  MoveL 3264 to (40.1, 47.39, -201.09) mm, rotated rx -152.51 ry -6.42 rz -112.51 deg; joints [11.465, -29.015, 82.683, 214.408, 104.039, 41.667, 26.033]
  MoveL 3265 to (39.93, 47.72, -201.04) mm, rotated rx -152.51 ry -6.42 rz -112.51 deg; joints [11.469, -29.014, 82.657, 214.407, 104.02, 41.65, 26.033]
  MoveL 3266 to (39.8, 48.12, -201) mm, rotated rx -152.51 ry -6.42 rz -112.51 deg; joints [11.471, -29.013, 82.629, 214.404, 103.997, 41.633, 26.033]
  MoveL 3267 to (39.72, 48.56, -200.98) mm, rotated rx -152.51 ry -6.42 rz -112.51 deg; joints [11.471, -29.014, 82.599, 214.4, 103.972, 41.615, 26.033]
  MoveL 3268 to (39.68, 49.06, -200.97) mm, rotated rx -152.51 ry -6.42 rz -112.51 deg; joints [11.47, -29.015, 82.566, 214.394, 103.943, 41.596, 26.033]
  MoveL 3269 to (39.66, 49.57, -200.97) mm, rotated rx -152.51 ry -6.42 rz -112.51 deg; joints [11.467, -29.017, 82.533, 214.388, 103.914, 41.577, 26.033]
  MoveL 3270 to (39.65, 50.63, -200.97) mm, rotated rx -152.51 ry -6.42 rz -112.51 deg; joints [11.461, -29.02, 82.466, 214.374, 103.854, 41.539, 26.033]
  MoveL 3271 to (39.63, 51.12, -200.95) mm, rotated rx -152.51 ry -6.42 rz -112.51 deg; joints [11.459, -29.021, 82.433, 214.368, 103.826, 41.52, 26.033]
  MoveL 3272 to (39.59, 51.58, -200.9) mm, rotated rx -152.51 ry -6.42 rz -112.51 deg; joints [11.458, -29.019, 82.399, 214.362, 103.798, 41.502, 26.033]
  MoveL 3273 to (39.53, 52.1, -200.82) mm, rotated rx -152.51 ry -6.42 rz -112.51 deg; joints [11.457, -29.016, 82.358, 214.357, 103.767, 41.481, 26.033]
  MoveL 3274 to (39.48, 52.68, -200.76) mm, rotated rx -152.51 ry -6.42 rz -112.51 deg; joints [11.456, -29.013, 82.315, 214.35, 103.733, 41.458, 26.033]
  MoveL 3275 to (39.45, 53.26, -200.73) mm, rotated rx -152.51 ry -6.42 rz -112.51 deg; joints [11.453, -29.013, 82.275, 214.343, 103.7, 41.436, 26.033]
  MoveL 3276 to (39.44, 53.79, -200.71) mm, rotated rx -152.51 ry -6.42 rz -112.51 deg; joints [11.45, -29.013, 82.239, 214.336, 103.669, 41.416, 26.033]
  MoveL 3277 to (39.43, 54.33, -200.71) mm, rotated rx -152.51 ry -6.42 rz -112.51 deg; joints [11.448, -29.015, 82.204, 214.329, 103.638, 41.397, 26.033]
  MoveL 3278 to (39.42, 55.38, -200.71) mm, rotated rx -152.51 ry -6.42 rz -112.51 deg; joints [11.442, -29.018, 82.137, 214.316, 103.578, 41.359, 26.033]
  MoveL 3279 to (39.37, 56.41, -200.69) mm, rotated rx -152.51 ry -6.42 rz -112.51 deg; joints [11.437, -29.019, 82.069, 214.303, 103.519, 41.321, 26.033]
  MoveL 3280 to (39.34, 59.03, -200.69) mm, rotated rx -152.51 ry -6.42 rz -112.51 deg; joints [11.423, -29.026, 81.9, 214.27, 103.369, 41.227, 26.033]
  MoveL 3281 to (39.39, 60.47, -200.77) mm, rotated rx -152.51 ry -6.42 rz -112.51 deg; joints [11.412, -29.035, 81.815, 214.25, 103.288, 41.178, 26.033]
  MoveL 3282 to (39.58, 61.64, -201.04) mm, rotated rx -152.51 ry -6.42 rz -112.51 deg; joints [11.398, -29.054, 81.764, 214.231, 103.225, 41.145, 26.033]
  MoveL 3283 to (39.9, 62.52, -201.47) mm, rotated rx -152.51 ry -6.42 rz -112.51 deg; joints [11.38, -29.083, 81.749, 214.213, 103.182, 41.128, 26.033]
  MoveL 3284 to (40.12, 62.85, -201.76) mm, rotated rx -152.51 ry -6.42 rz -112.51 deg; joints [11.37, -29.102, 81.754, 214.204, 103.168, 41.126, 26.033]
  MoveL 3285 to (40.37, 63.12, -202.09) mm, rotated rx -152.51 ry -6.42 rz -112.51 deg; joints [11.359, -29.123, 81.768, 214.196, 103.158, 41.128, 26.033]
  MoveL 3286 to (40.97, 63.44, -202.88) mm, rotated rx -152.51 ry -6.42 rz -112.51 deg; joints [11.334, -29.173, 81.823, 214.179, 103.153, 41.143, 26.033]
  MoveL 3287 to (41.71, 63.48, -203.84) mm, rotated rx -152.51 ry -6.42 rz -112.51 deg; joints [11.305, -29.234, 81.912, 214.164, 103.167, 41.174, 26.033]
  MoveL 3288 to (43.6, 62.7, -206.3) mm, rotated rx -152.51 ry -6.42 rz -112.51 deg; joints [11.236, -29.386, 82.195, 214.134, 103.252, 41.285, 26.033]
  MoveL 3289 to (45.46, 61.14, -208.75) mm, rotated rx -152.51 ry -6.42 rz -112.51 deg; joints [11.173, -29.535, 82.528, 214.116, 103.383, 41.423, 26.033]
  MoveL 3290 to (46.69, 59.12, -210.51) mm, rotated rx -152.51 ry -6.42 rz -112.51 deg; joints [11.137, -29.64, 82.823, 214.117, 103.527, 41.551, 26.033]
  MoveL 3291 to (47.06, 57.94, -211.12) mm, rotated rx -152.51 ry -6.42 rz -112.51 deg; joints [11.129, -29.676, 82.957, 214.124, 103.605, 41.612, 26.033]
  MoveL 3292 to (47.28, 56.65, -211.56) mm, rotated rx -152.51 ry -6.42 rz -112.51 deg; joints [11.127, -29.701, 83.081, 214.137, 103.687, 41.67, 26.033]
  MoveL 3293 to (47.24, 53.72, -211.91) mm, rotated rx -152.51 ry -6.42 rz -112.51 deg; joints [11.144, -29.717, 83.301, 214.176, 103.862, 41.78, 26.033]
  MoveL 3294 to (46.95, 51.11, -211.91) mm, rotated rx -152.51 ry -6.42 rz -112.51 deg; joints [11.169, -29.712, 83.467, 214.217, 104.012, 41.867, 26.033]
  MoveL 3295 to (46.88, 50.59, -211.9) mm, rotated rx -152.51 ry -6.42 rz -112.51 deg; joints [11.174, -29.71, 83.5, 214.226, 104.042, 41.884, 26.033]
  MoveL 3296 to (46.8, 50.05, -211.87) mm, rotated rx -152.51 ry -6.42 rz -112.51 deg; joints [11.18, -29.707, 83.531, 214.235, 104.073, 41.901, 26.033]
  MoveL 3297 to (46.74, 49.56, -211.86) mm, rotated rx -152.51 ry -6.42 rz -112.51 deg; joints [11.185, -29.705, 83.561, 214.243, 104.101, 41.917, 26.033]
  MoveL 3298 to (46.7, 49.11, -211.88) mm, rotated rx -152.51 ry -6.42 rz -112.51 deg; joints [11.189, -29.705, 83.591, 214.249, 104.127, 41.932, 26.033]
  MoveL 3299 to (46.66, 48.63, -211.9) mm, rotated rx -152.51 ry -6.42 rz -112.51 deg; joints [11.193, -29.706, 83.625, 214.257, 104.155, 41.949, 26.033]
  MoveL 3300 to (46.64, 48.05, -211.97) mm, rotated rx -152.51 ry -6.42 rz -112.51 deg; joints [11.197, -29.709, 83.668, 214.265, 104.19, 41.97, 26.033]
  MoveL 3301 to (46.63, 47.47, -212.05) mm, rotated rx -152.51 ry -6.42 rz -112.51 deg; joints [11.2, -29.712, 83.711, 214.273, 104.224, 41.992, 26.033]
  MoveL 3302 to (46.6, 46.9, -212.1) mm, rotated rx -152.51 ry -6.42 rz -112.51 deg; joints [11.204, -29.714, 83.752, 214.282, 104.257, 42.013, 26.033]
  MoveL 3303 to (46.56, 46.37, -212.12) mm, rotated rx -152.51 ry -6.42 rz -112.51 deg; joints [11.209, -29.714, 83.787, 214.29, 104.288, 42.031, 26.033]
  MoveL 3304 to (46.5, 45.86, -212.13) mm, rotated rx -152.51 ry -6.42 rz -112.51 deg; joints [11.214, -29.713, 83.821, 214.298, 104.318, 42.048, 26.033]
  MoveL 3305 to (46.45, 45.34, -212.13) mm, rotated rx -152.51 ry -6.42 rz -112.51 deg; joints [11.219, -29.712, 83.854, 214.306, 104.348, 42.066, 26.033]
  MoveL 3306 to (46.41, 44.77, -212.16) mm, rotated rx -152.51 ry -6.42 rz -112.51 deg; joints [11.223, -29.712, 83.892, 214.315, 104.381, 42.086, 26.033]
  MoveL 3307 to (46.39, 44.22, -212.22) mm, rotated rx -152.51 ry -6.42 rz -112.51 deg; joints [11.227, -29.714, 83.932, 214.323, 104.413, 42.106, 26.033]
  MoveL 3308 to (46.39, 43.66, -212.29) mm, rotated rx -152.51 ry -6.42 rz -112.51 deg; joints [11.23, -29.717, 83.973, 214.331, 104.446, 42.127, 26.033]
  MoveL 3309 to (46.45, 43.16, -212.35) mm, rotated rx -152.51 ry -6.42 rz -112.51 deg; joints [11.231, -29.718, 84.01, 214.336, 104.476, 42.147, 26.033]
  MoveL 3310 to (46.54, 42.71, -212.38) mm, rotated rx -152.51 ry -6.42 rz -112.51 deg; joints [11.23, -29.718, 84.041, 214.341, 104.502, 42.166, 26.033]
  MoveL 3311 to (46.68, 42.33, -212.39) mm, rotated rx -152.51 ry -6.42 rz -112.51 deg; joints [11.227, -29.715, 84.066, 214.343, 104.523, 42.183, 26.033]
  MoveL 3312 to (46.84, 41.98, -212.39) mm, rotated rx -152.51 ry -6.42 rz -112.51 deg; joints [11.224, -29.712, 84.087, 214.344, 104.542, 42.199, 26.033]
  MoveL 3313 to (46.45, 43.21, -213.26) mm, rotated rx -152.51 ry -6.42 rz -112.51 deg; joints [11.226, -29.782, 84.094, 214.336, 104.491, 42.161, 26.033]
  MoveL 3314 to (47.29, 41.84, -213.54) mm, rotated rx -152.51 ry -6.42 rz -112.51 deg; joints [11.205, -29.787, 84.204, 214.337, 104.57, 42.233, 26.033]
  MoveL 3315 to (48.19, 40.28, -213.74) mm, rotated rx -152.51 ry -6.42 rz -112.51 deg; joints [11.183, -29.785, 84.318, 214.339, 104.66, 42.311, 26.033]
  MoveL 3316 to (49.17, 38.48, -213.87) mm, rotated rx -152.51 ry -6.42 rz -112.51 deg; joints [11.161, -29.777, 84.441, 214.343, 104.761, 42.399, 26.033]
  MoveL 3317 to (50.22, 36.49, -213.96) mm, rotated rx -152.51 ry -6.42 rz -112.51 deg; joints [11.137, -29.763, 84.571, 214.348, 104.871, 42.494, 26.033]
  MoveL 3318 to (51.24, 34.61, -214.11) mm, rotated rx -152.51 ry -6.42 rz -112.51 deg; joints [11.114, -29.754, 84.699, 214.353, 104.976, 42.586, 26.033]
  MoveL 3319 to (52.26, 32.73, -214.32) mm, rotated rx -152.51 ry -6.42 rz -112.51 deg; joints [11.09, -29.749, 84.832, 214.357, 105.083, 42.678, 26.033]
  MoveL 3320 to (53.22, 30.94, -214.44) mm, rotated rx -152.51 ry -6.42 rz -112.51 deg; joints [11.068, -29.739, 84.951, 214.362, 105.183, 42.765, 26.033]
  MoveL 3321 to (54.11, 29.32, -214.71) mm, rotated rx -152.51 ry -6.42 rz -112.51 deg; joints [11.046, -29.739, 85.073, 214.365, 105.276, 42.846, 26.033]
  MoveL 3322 to (55.08, 27.5, -214.92) mm, rotated rx -152.51 ry -6.42 rz -112.51 deg; joints [11.024, -29.735, 85.202, 214.37, 105.379, 42.935, 26.033]
  MoveL 3323 to (56.05, 25.66, -215.06) mm, rotated rx -152.51 ry -6.42 rz -112.51 deg; joints [11.001, -29.724, 85.325, 214.375, 105.482, 43.024, 26.033]
  MoveL 3324 to (57.04, 23.77, -215.17) mm, rotated rx -152.51 ry -6.42 rz -112.51 deg; joints [10.979, -29.71, 85.447, 214.381, 105.587, 43.115, 26.033]
  MoveL 3325 to (58.04, 21.89, -215.4) mm, rotated rx -152.51 ry -6.42 rz -112.51 deg; joints [10.956, -29.705, 85.579, 214.387, 105.693, 43.207, 26.033]
  MoveL 3326 to (59.01, 19.98, -215.66) mm, rotated rx -152.51 ry -6.42 rz -112.51 deg; joints [10.933, -29.701, 85.716, 214.393, 105.802, 43.3, 26.033]
  MoveL 3327 to (59.99, 18.09, -215.74) mm, rotated rx -152.51 ry -6.42 rz -112.51 deg; joints [10.911, -29.685, 85.835, 214.399, 105.906, 43.39, 26.033]
  MoveL 3328 to (60.99, 16.16, -215.79) mm, rotated rx -152.51 ry -6.42 rz -112.51 deg; joints [10.888, -29.666, 85.952, 214.406, 106.012, 43.481, 26.033]
  MoveL 3329 to (61.95, 14.28, -215.89) mm, rotated rx -152.51 ry -6.42 rz -112.51 deg; joints [10.867, -29.651, 86.071, 214.412, 106.116, 43.57, 26.033]
  MoveL 3330 to (62.91, 12.39, -216.1) mm, rotated rx -152.51 ry -6.42 rz -112.51 deg; joints [10.844, -29.642, 86.2, 214.419, 106.222, 43.662, 26.033]
  MoveL 3331 to (63.84, 10.53, -216.43) mm, rotated rx -152.51 ry -6.42 rz -112.51 deg; joints [10.822, -29.642, 86.338, 214.426, 106.329, 43.753, 26.033]
  MoveL 3332 to (64.79, 8.6, -216.69) mm, rotated rx -152.51 ry -6.42 rz -112.51 deg; joints [10.801, -29.637, 86.474, 214.435, 106.439, 43.847, 26.033]
  MoveL 3333 to (65.73, 6.68, -216.89) mm, rotated rx -152.51 ry -6.42 rz -112.51 deg; joints [10.779, -29.627, 86.602, 214.443, 106.547, 43.939, 26.033]
  MoveL 3334 to (66.67, 4.72, -217.13) mm, rotated rx -152.51 ry -6.42 rz -112.51 deg; joints [10.758, -29.619, 86.737, 214.452, 106.657, 44.033, 26.033]
  MoveL 3335 to (67.63, 2.79, -217.27) mm, rotated rx -152.51 ry -6.42 rz -112.51 deg; joints [10.736, -29.604, 86.86, 214.46, 106.764, 44.124, 26.033]
  MoveL 3336 to (68.6, 0.91, -217.29) mm, rotated rx -152.51 ry -6.42 rz -112.51 deg; joints [10.714, -29.581, 86.968, 214.467, 106.866, 44.212, 26.033]
  MoveL 3337 to (68.51, 0.28, -217.96) mm, rotated rx -152.51 ry -6.42 rz -112.51 deg; joints [10.717, -29.622, 87.067, 214.479, 106.914, 44.244, 26.033]
  MoveL 3338 to (68.29, 0.53, -218.29) mm, rotated rx -152.51 ry -6.42 rz -112.51 deg; joints [10.722, -29.649, 87.083, 214.48, 106.908, 44.236, 26.033]
  MoveL 3339 to (68.26, 0.56, -218.49) mm, rotated rx -152.51 ry -6.42 rz -112.51 deg; joints [10.722, -29.663, 87.101, 214.481, 106.91, 44.238, 26.033]
  MoveL 3340 to (68.4, 0.39, -218.59) mm, rotated rx -152.51 ry -6.42 rz -112.51 deg; joints [10.718, -29.668, 87.12, 214.48, 106.921, 44.249, 26.033]
  MoveL 3341 to (68.72, 0.12, -218.62) mm, rotated rx -152.51 ry -6.42 rz -112.51 deg; joints [10.708, -29.663, 87.137, 214.477, 106.935, 44.266, 26.033]
  MoveC 3342 to (69.58, -0.43, -218.62) mm, rotated rx -152.51 ry -6.42 rz -112.51 deg; joints [10.682, -29.65, 87.166, 214.466, 106.963, 44.303, 26.033] to (70.47, -0.92, -218.62) mm, rotated rx -152.51 ry -6.42 rz -112.51 deg; joints [10.655, -29.636, 87.191, 214.454, 106.986, 44.338, 26.033]
  MoveL 3343 to (70.47, -0.92, -218.62) mm, rotated rx -152.51 ry -6.42 rz -112.51 deg; joints [10.655, -29.636, 87.191, 214.454, 106.987, 44.339, 26.033]
  MoveL 3344 to (70.94, -1.19, -218.64) mm, rotated rx -152.51 ry -6.42 rz -112.51 deg; joints [10.641, -29.631, 87.208, 214.447, 107, 44.358, 26.033]
  MoveL 3345 to (71.39, -1.48, -218.69) mm, rotated rx -152.51 ry -6.42 rz -112.51 deg; joints [10.627, -29.627, 87.227, 214.441, 107.015, 44.379, 26.033]
  MoveL 3346 to (71.88, -1.79, -218.76) mm, rotated rx -152.51 ry -6.42 rz -112.51 deg; joints [10.612, -29.623, 87.25, 214.435, 107.033, 44.401, 26.033]
  MoveL 3347 to (72.39, -2.1, -218.8) mm, rotated rx -152.51 ry -6.42 rz -112.51 deg; joints [10.596, -29.618, 87.27, 214.429, 107.049, 44.423, 26.033]
  MoveL 3348 to (73.45, -2.7, -218.82) mm, rotated rx -152.51 ry -6.42 rz -112.51 deg; joints [10.563, -29.603, 87.303, 214.414, 107.078, 44.467, 26.033]
  MoveL 3349 to (73.92, -2.99, -218.86) mm, rotated rx -152.51 ry -6.42 rz -112.51 deg; joints [10.549, -29.598, 87.321, 214.408, 107.093, 44.487, 26.033]
  MoveL 3350 to (74.31, -3.26, -218.93) mm, rotated rx -152.51 ry -6.42 rz -112.51 deg; joints [10.537, -29.596, 87.342, 214.403, 107.108, 44.506, 26.033]
  MoveL 3351 to (74.67, -3.52, -219.02) mm, rotated rx -152.51 ry -6.42 rz -112.51 deg; joints [10.526, -29.596, 87.364, 214.399, 107.123, 44.524, 26.033]
  MoveL 3352 to (75.02, -3.75, -219.08) mm, rotated rx -152.51 ry -6.42 rz -112.51 deg; joints [10.515, -29.595, 87.382, 214.395, 107.136, 44.541, 26.033]
  MoveL 3353 to (75.4, -3.99, -219.12) mm, rotated rx -152.51 ry -6.42 rz -112.51 deg; joints [10.503, -29.591, 87.398, 214.39, 107.148, 44.557, 26.033]
  MoveL 3354 to (77.7, -5.25, -219.12) mm, rotated rx -152.51 ry -6.42 rz -112.51 deg; joints [10.433, -29.555, 87.461, 214.357, 107.209, 44.649, 26.033]
  MoveL 3355 to (80.11, -6.88, -219.46) mm, rotated rx -152.51 ry -6.42 rz -112.51 deg; joints [10.358, -29.538, 87.577, 214.327, 107.297, 44.762, 26.033]
  MoveL 3356 to (81.03, -7.77, -219.89) mm, rotated rx -152.51 ry -6.42 rz -112.51 deg; joints [10.33, -29.549, 87.665, 214.321, 107.351, 44.819, 26.033]
  MoveL 3357 to (81.76, -8.71, -220.5) mm, rotated rx -152.51 ry -6.42 rz -112.51 deg; joints [10.307, -29.573, 87.771, 214.319, 107.413, 44.878, 26.033]
  MoveL 3358 to (82.31, -9.71, -221.27) mm, rotated rx -152.51 ry -6.42 rz -112.51 deg; joints [10.291, -29.611, 87.897, 214.323, 107.481, 44.938, 26.033]
  MoveL 3359 to (82.67, -10.76, -222.22) mm, rotated rx -152.51 ry -6.42 rz -112.51 deg; joints [10.28, -29.662, 88.043, 214.332, 107.556, 44.999, 26.033]
  MoveL 3360 to (82.82, -13.01, -224.64) mm, rotated rx -152.51 ry -6.42 rz -112.51 deg; joints [10.275, -29.803, 88.392, 214.366, 107.726, 45.124, 26.033]
  MoveL 3361 to (82.3, -14.84, -227.05) mm, rotated rx -152.51 ry -6.42 rz -112.51 deg; joints [10.291, -29.955, 88.719, 214.409, 107.874, 45.221, 26.033]
  MoveL 3362 to (81.82, -15.37, -228) mm, rotated rx -152.51 ry -6.42 rz -112.51 deg; joints [10.306, -30.02, 88.836, 214.429, 107.923, 45.246, 26.033]
  MoveL 3363 to (81.19, -15.62, -228.77) mm, rotated rx -152.51 ry -6.42 rz -112.51 deg; joints [10.325, -30.077, 88.924, 214.448, 107.954, 45.256, 26.033]
  MoveL 3364 to (80.82, -15.65, -229.1) mm, rotated rx -152.51 ry -6.42 rz -112.51 deg; joints [10.336, -30.103, 88.957, 214.458, 107.963, 45.255, 26.033]
  MoveL 3365 to (80.41, -15.62, -229.38) mm, rotated rx -152.51 ry -6.42 rz -112.51 deg; joints [10.348, -30.126, 88.982, 214.467, 107.968, 45.25, 26.033]
  MoveL 3366 to (79.49, -15.35, -229.81) mm, rotated rx -152.51 ry -6.42 rz -112.51 deg; joints [10.376, -30.168, 89.01, 214.484, 107.964, 45.229, 26.033]
  MoveL 3367 to (78.42, -14.82, -230.07) mm, rotated rx -152.51 ry -6.42 rz -112.51 deg; joints [10.408, -30.203, 89.008, 214.5, 107.943, 45.193, 26.033]
  MoveL 3368 to (77.21, -14.03, -230.15) mm, rotated rx -152.51 ry -6.42 rz -112.51 deg; joints [10.445, -30.23, 88.975, 214.516, 107.905, 45.141, 26.033]
  MoveL 3369 to (76.78, -13.72, -230.15) mm, rotated rx -152.51 ry -6.42 rz -112.51 deg; joints [10.458, -30.237, 88.96, 214.521, 107.89, 45.122, 26.033]
  MoveL 3370 to (76.43, -13.44, -230.12) mm, rotated rx -152.51 ry -6.42 rz -112.51 deg; joints [10.468, -30.241, 88.942, 214.524, 107.875, 45.104, 26.033]
  MoveL 3371 to (76.11, -13.17, -230.07) mm, rotated rx -152.51 ry -6.42 rz -112.51 deg; joints [10.478, -30.244, 88.923, 214.527, 107.86, 45.087, 26.033]
  MoveL 3372 to (75.8, -12.9, -229.99) mm, rotated rx -152.51 ry -6.42 rz -112.51 deg; joints [10.487, -30.245, 88.902, 214.53, 107.845, 45.069, 26.033]
  MoveL 3373 to (75.46, -12.61, -229.95) mm, rotated rx -152.51 ry -6.42 rz -112.51 deg; joints [10.497, -30.248, 88.883, 214.533, 107.83, 45.052, 26.033]
  MoveL 3374 to (75.06, -12.31, -229.93) mm, rotated rx -152.51 ry -6.42 rz -112.51 deg; joints [10.509, -30.254, 88.866, 214.538, 107.814, 45.032, 26.033]
  MoveL 3375 to (70.41, -8.97, -229.92) mm, rotated rx -152.51 ry -6.42 rz -112.51 deg; joints [10.649, -30.335, 88.691, 214.591, 107.645, 44.817, 26.033]
  MoveL 3376 to (69.79, -8.51, -229.91) mm, rotated rx -152.51 ry -6.42 rz -112.51 deg; joints [10.667, -30.345, 88.666, 214.598, 107.621, 44.788, 26.033]
  MoveL 3377 to (69.28, -8.09, -229.9) mm, rotated rx -152.51 ry -6.42 rz -112.51 deg; joints [10.682, -30.354, 88.643, 214.603, 107.6, 44.762, 26.033]
  MoveL 3378 to (68.9, -7.66, -229.89) mm, rotated rx -152.51 ry -6.42 rz -112.51 deg; joints [10.693, -30.361, 88.619, 214.605, 107.577, 44.739, 26.033]
  MoveL 3379 to (68.6, -7.22, -229.85) mm, rotated rx -152.51 ry -6.42 rz -112.51 deg; joints [10.701, -30.365, 88.591, 214.604, 107.553, 44.716, 26.033]
  MoveL 3380 to (68.46, -6.92, -229.69) mm, rotated rx -152.51 ry -6.42 rz -112.51 deg; joints [10.704, -30.358, 88.559, 214.603, 107.533, 44.699, 26.033]
  MoveL 3381 to (68.48, -6.9, -229.38) mm, rotated rx -152.51 ry -6.42 rz -112.51 deg; joints [10.705, -30.337, 88.53, 214.602, 107.527, 44.694, 26.033]
  MoveL 3382 to (68.68, -7.21, -228.89) mm, rotated rx -152.51 ry -6.42 rz -112.51 deg; joints [10.703, -30.3, 88.503, 214.602, 107.535, 44.701, 26.033]
  MoveL 3383 to (69.07, -6.72, -227.92) mm, rotated rx -152.51 ry -6.42 rz -112.51 deg; joints [10.691, -30.234, 88.385, 214.584, 107.488, 44.676, 26.033]
  MoveL 3384 to (68.45, -4.96, -227.62) mm, rotated rx -152.51 ry -6.42 rz -112.51 deg; joints [10.703, -30.235, 88.258, 214.57, 107.387, 44.594, 26.033]
  MoveL 3385 to (67.8, -3.11, -227.41) mm, rotated rx -152.51 ry -6.42 rz -112.51 deg; joints [10.716, -30.244, 88.135, 214.556, 107.282, 44.51, 26.033]
  MoveL 3386 to (67.07, -1.11, -227.29) mm, rotated rx -152.51 ry -6.42 rz -112.51 deg; joints [10.729, -30.259, 88.011, 214.541, 107.171, 44.421, 26.033]
  MoveL 3387 to (65.57, 2.89, -227.29) mm, rotated rx -152.51 ry -6.42 rz -112.51 deg; joints [10.756, -30.307, 87.783, 214.512, 106.953, 44.245, 26.033]
  MoveL 3388 to (64.88, 4.75, -227.2) mm, rotated rx -152.51 ry -6.42 rz -112.51 deg; joints [10.769, -30.322, 87.669, 214.499, 106.85, 44.162, 26.033]
  MoveL 3389 to (64.13, 6.74, -227.2) mm, rotated rx -152.51 ry -6.42 rz -112.51 deg; joints [10.783, -30.345, 87.554, 214.485, 106.741, 44.075, 26.033]
  MoveL 3390 to (63.47, 8.8, -227.2) mm, rotated rx -152.51 ry -6.42 rz -112.51 deg; joints [10.793, -30.367, 87.436, 214.468, 106.628, 43.987, 26.033]
  MoveL 3391 to (62.73, 11.23, -227.02) mm, rotated rx -152.51 ry -6.42 rz -112.51 deg; joints [10.805, -30.38, 87.278, 214.448, 106.491, 43.881, 26.033]
  MoveL 3392 to (61.83, 13.27, -226.79) mm, rotated rx -152.51 ry -6.42 rz -112.51 deg; joints [10.825, -30.388, 87.139, 214.437, 106.376, 43.785, 26.033]
  MoveL 3393 to (60.98, 15.27, -226.67) mm, rotated rx -152.51 ry -6.42 rz -112.51 deg; joints [10.842, -30.402, 87.012, 214.426, 106.264, 43.693, 26.033]
  MoveL 3394 to (60.23, 17.27, -226.56) mm, rotated rx -152.51 ry -6.42 rz -112.51 deg; joints [10.856, -30.416, 86.885, 214.413, 106.153, 43.604, 26.033]
  MoveL 3395 to (59.47, 19.26, -226.34) mm, rotated rx -152.51 ry -6.42 rz -112.51 deg; joints [10.871, -30.422, 86.748, 214.4, 106.039, 43.512, 26.033]
  MoveL 3396 to (58.72, 21.26, -226.24) mm, rotated rx -152.51 ry -6.42 rz -112.51 deg; joints [10.885, -30.435, 86.62, 214.387, 105.928, 43.423, 26.033]
  MoveL 3397 to (57.97, 23.26, -226.13) mm, rotated rx -152.51 ry -6.42 rz -112.51 deg; joints [10.899, -30.448, 86.492, 214.374, 105.816, 43.334, 26.033]
  MoveL 3398 to (57.2, 25.25, -225.91) mm, rotated rx -152.51 ry -6.42 rz -112.51 deg; joints [10.914, -30.453, 86.354, 214.362, 105.703, 43.243, 26.033]
  MoveL 3399 to (56.44, 27.24, -225.81) mm, rotated rx -152.51 ry -6.42 rz -112.51 deg; joints [10.929, -30.465, 86.226, 214.35, 105.591, 43.153, 26.033]
  MoveL 3400 to (55.68, 29.23, -225.7) mm, rotated rx -152.51 ry -6.42 rz -112.51 deg; joints [10.943, -30.477, 86.097, 214.338, 105.48, 43.064, 26.033]
  MoveL 3401 to (54.9, 31.22, -225.5) mm, rotated rx -152.51 ry -6.42 rz -112.51 deg; joints [10.958, -30.482, 85.959, 214.326, 105.366, 42.973, 26.033]
  MoveL 3402 to (54.13, 33.21, -225.4) mm, rotated rx -152.51 ry -6.42 rz -112.51 deg; joints [10.973, -30.493, 85.829, 214.315, 105.255, 42.883, 26.033]
  MoveL 3403 to (53.4, 34.91, -225.14) mm, rotated rx -152.51 ry -6.42 rz -112.51 deg; joints [10.989, -30.492, 85.703, 214.306, 105.156, 42.803, 26.033]
  MoveL 3404 to (52.68, 36.42, -224.77) mm, rotated rx -152.51 ry -6.42 rz -112.51 deg; joints [11.005, -30.481, 85.578, 214.301, 105.067, 42.728, 26.033]
  MoveL 3405 to (51.97, 37.76, -224.27) mm, rotated rx -152.51 ry -6.42 rz -112.51 deg; joints [11.024, -30.461, 85.45, 214.297, 104.984, 42.656, 26.033]
  MoveL 3406 to (52.12, 36.64, -223.43) mm, rotated rx -152.51 ry -6.42 rz -112.51 deg; joints [11.029, -30.396, 85.441, 214.309, 105.032, 42.686, 26.033]
  MoveL 3407 to (52.01, 36.95, -223.4) mm, rotated rx -152.51 ry -6.42 rz -112.51 deg; joints [11.031, -30.397, 85.419, 214.307, 105.014, 42.672, 26.033]
  MoveL 3408 to (51.93, 37.26, -223.35) mm, rotated rx -152.51 ry -6.42 rz -112.51 deg; joints [11.032, -30.396, 85.396, 214.305, 104.996, 42.658, 26.033]
  MoveL 3409 to (51.91, 37.63, -223.3) mm, rotated rx -152.51 ry -6.42 rz -112.51 deg; joints [11.031, -30.394, 85.368, 214.3, 104.974, 42.644, 26.033]
  MoveL 3410 to (51.95, 38.05, -223.26) mm, rotated rx -152.51 ry -6.42 rz -112.51 deg; joints [11.027, -30.393, 85.339, 214.293, 104.95, 42.629, 26.033]
  MoveL 3411 to (52.03, 38.52, -223.24) mm, rotated rx -152.51 ry -6.42 rz -112.51 deg; joints [11.022, -30.393, 85.307, 214.285, 104.922, 42.613, 26.033]
  MoveL 3412 to (53.12, 43.11, -223.24) mm, rotated rx -152.51 ry -6.42 rz -112.51 deg; joints [10.959, -30.402, 85.021, 214.197, 104.657, 42.472, 26.033]
  MoveL 3413 to (53.19, 43.5, -223.21) mm, rotated rx -152.51 ry -6.42 rz -112.51 deg; joints [10.954, -30.401, 84.993, 214.19, 104.634, 42.459, 26.033]
  MoveL 3414 to (53.31, 44.01, -223.21) mm, rotated rx -152.51 ry -6.42 rz -112.51 deg; joints [10.947, -30.402, 84.961, 214.18, 104.604, 42.444, 26.033]
  MoveL 3415 to (53.52, 45.02, -223.17) mm, rotated rx -152.51 ry -6.42 rz -112.51 deg; joints [10.934, -30.401, 84.894, 214.162, 104.545, 42.412, 26.033]
  MoveL 3416 to (54.13, 47.57, -223.17) mm, rotated rx -152.51 ry -6.42 rz -112.51 deg; joints [10.899, -30.405, 84.734, 214.114, 104.397, 42.333, 26.033]
  MoveL 3417 to (54.31, 48.58, -223.15) mm, rotated rx -152.51 ry -6.42 rz -112.51 deg; joints [10.888, -30.406, 84.668, 214.096, 104.338, 42.301, 26.033]
  MoveL 3418 to (54.62, 50, -223.22) mm, rotated rx -152.51 ry -6.42 rz -112.51 deg; joints [10.869, -30.413, 84.585, 214.07, 104.258, 42.258, 26.033]
  MoveL 3419 to (55.02, 51.1, -223.47) mm, rotated rx -152.51 ry -6.42 rz -112.51 deg; joints [10.848, -30.43, 84.538, 214.047, 104.198, 42.232, 26.033]
  MoveL 3420 to (55.49, 51.9, -223.91) mm, rotated rx -152.51 ry -6.42 rz -112.51 deg; joints [10.825, -30.458, 84.527, 214.026, 104.158, 42.22, 26.033]
  MoveL 3421 to (55.76, 52.18, -224.2) mm, rotated rx -152.51 ry -6.42 rz -112.51 deg; joints [10.814, -30.477, 84.536, 214.016, 104.146, 42.221, 26.033]
  MoveL 3422 to (56.04, 52.39, -224.54) mm, rotated rx -152.51 ry -6.42 rz -112.51 deg; joints [10.801, -30.498, 84.553, 214.007, 104.139, 42.225, 26.033]
  MoveL 3423 to (56.67, 52.58, -225.35) mm, rotated rx -152.51 ry -6.42 rz -112.51 deg; joints [10.775, -30.548, 84.615, 213.991, 104.141, 42.245, 26.033]
  MoveL 3424 to (57.38, 52.46, -226.35) mm, rotated rx -152.51 ry -6.42 rz -112.51 deg; joints [10.748, -30.609, 84.714, 213.978, 104.163, 42.28, 26.033]
  MoveL 3425 to (59.03, 51.31, -228.91) mm, rotated rx -152.51 ry -6.42 rz -112.51 deg; joints [10.687, -30.764, 85.019, 213.957, 104.268, 42.397, 26.033]
  MoveL 3426 to (60.48, 49.4, -231.47) mm, rotated rx -152.51 ry -6.42 rz -112.51 deg; joints [10.637, -30.917, 85.373, 213.952, 104.417, 42.537, 26.033]
  MoveL 3427 to (61.2, 47.18, -233.3) mm, rotated rx -152.51 ry -6.42 rz -112.51 deg; joints [10.617, -31.026, 85.678, 213.966, 104.574, 42.661, 26.033]
  MoveL 3428 to (61.29, 45.96, -233.94) mm, rotated rx -152.51 ry -6.42 rz -112.51 deg; joints [10.618, -31.064, 85.813, 213.981, 104.655, 42.716, 26.033]
  MoveL 3429 to (61.2, 44.66, -234.4) mm, rotated rx -152.51 ry -6.42 rz -112.51 deg; joints [10.627, -31.091, 85.936, 214.001, 104.737, 42.768, 26.033]
  MoveL 3430 to (60.47, 41.83, -234.77) mm, rotated rx -152.51 ry -6.42 rz -112.51 deg; joints [10.665, -31.11, 86.147, 214.056, 104.908, 42.859, 26.033]
  MoveL 3431 to (59.39, 38.87, -234.77) mm, rotated rx -152.51 ry -6.42 rz -112.51 deg; joints [10.719, -31.108, 86.331, 214.121, 105.08, 42.942, 26.033]
  MoveL 3432 to (59.06, 37.91, -234.78) mm, rotated rx -152.51 ry -6.42 rz -112.51 deg; joints [10.735, -31.107, 86.393, 214.142, 105.136, 42.97, 26.033]
  MoveL 3433 to (58.7, 36.93, -234.78) mm, rotated rx -152.51 ry -6.42 rz -112.51 deg; joints [10.753, -31.106, 86.454, 214.164, 105.194, 42.997, 26.033]
  MoveL 3434 to (58.54, 36.46, -234.79) mm, rotated rx -152.51 ry -6.42 rz -112.51 deg; joints [10.761, -31.106, 86.484, 214.174, 105.221, 43.011, 26.033]
  MoveL 3435 to (58.32, 35.83, -234.82) mm, rotated rx -152.51 ry -6.42 rz -112.51 deg; joints [10.772, -31.107, 86.525, 214.188, 105.258, 43.029, 26.033]
  MoveL 3436 to (58.14, 35.26, -234.87) mm, rotated rx -152.51 ry -6.42 rz -112.51 deg; joints [10.781, -31.11, 86.566, 214.2, 105.292, 43.046, 26.033]
  MoveL 3437 to (58.01, 34.77, -234.95) mm, rotated rx -152.51 ry -6.42 rz -112.51 deg; joints [10.788, -31.114, 86.602, 214.21, 105.322, 43.062, 26.033]
  MoveL 3438 to (57.88, 34.33, -235) mm, rotated rx -152.51 ry -6.42 rz -112.51 deg; joints [10.795, -31.116, 86.635, 214.219, 105.348, 43.076, 26.033]
  MoveL 3439 to (57.74, 33.88, -235.03) mm, rotated rx -152.51 ry -6.42 rz -112.51 deg; joints [10.802, -31.118, 86.665, 214.228, 105.375, 43.09, 26.033]
  MoveL 3440 to (57.21, 32.41, -235.03) mm, rotated rx -152.51 ry -6.42 rz -112.51 deg; joints [10.829, -31.115, 86.756, 214.262, 105.46, 43.131, 26.033]
  MoveL 3441 to (57.05, 31.93, -235.05) mm, rotated rx -152.51 ry -6.42 rz -112.51 deg; joints [10.837, -31.115, 86.787, 214.272, 105.488, 43.146, 26.033]
  MoveL 3442 to (56.94, 31.51, -235.07) mm, rotated rx -152.51 ry -6.42 rz -112.51 deg; joints [10.843, -31.116, 86.816, 214.28, 105.513, 43.159, 26.033]
  MoveL 3443 to (56.87, 31.13, -235.12) mm, rotated rx -152.51 ry -6.42 rz -112.51 deg; joints [10.847, -31.118, 86.843, 214.288, 105.536, 43.172, 26.033]
  MoveL 3444 to (56.88, 30.82, -235.19) mm, rotated rx -152.51 ry -6.42 rz -112.51 deg; joints [10.848, -31.121, 86.868, 214.292, 105.554, 43.184, 26.033]
  MoveL 3445 to (56.93, 30.55, -235.26) mm, rotated rx -152.51 ry -6.42 rz -112.51 deg; joints [10.848, -31.123, 86.89, 214.295, 105.571, 43.196, 26.033]
  MoveL 3446 to (57.25, 32.11, -236.06) mm, rotated rx -152.51 ry -6.42 rz -112.51 deg; joints [10.824, -31.183, 86.868, 214.265, 105.495, 43.159, 26.033]
  MoveL 3447 to (57.63, 30.38, -236.46) mm, rotated rx -152.51 ry -6.42 rz -112.51 deg; joints [10.819, -31.197, 87.009, 214.282, 105.599, 43.236, 26.033]
  MoveL 3448 to (58.06, 28.56, -236.73) mm, rotated rx -152.51 ry -6.42 rz -112.51 deg; joints [10.814, -31.2, 87.142, 214.299, 105.705, 43.315, 26.033]
  MoveL 3449 to (58.55, 26.62, -236.91) mm, rotated rx -152.51 ry -6.42 rz -112.51 deg; joints [10.808, -31.196, 87.275, 214.316, 105.816, 43.398, 26.033]
  MoveL 3450 to (59.09, 24.55, -237.1) mm, rotated rx -152.51 ry -6.42 rz -112.51 deg; joints [10.801, -31.191, 87.415, 214.335, 105.934, 43.486, 26.033]
  MoveL 3451 to (59.62, 22.48, -237.2) mm, rotated rx -152.51 ry -6.42 rz -112.51 deg; joints [10.795, -31.179, 87.547, 214.354, 106.05, 43.573, 26.033]
  MoveL 3452 to (60.13, 20.41, -237.3) mm, rotated rx -152.51 ry -6.42 rz -112.51 deg; joints [10.789, -31.167, 87.678, 214.373, 106.167, 43.66, 26.033]
  MoveL 3453 to (60.66, 18.35, -237.49) mm, rotated rx -152.51 ry -6.42 rz -112.51 deg; joints [10.783, -31.161, 87.818, 214.392, 106.285, 43.749, 26.033]
  MoveL 3454 to (61.18, 16.28, -237.59) mm, rotated rx -152.51 ry -6.42 rz -112.51 deg; joints [10.777, -31.148, 87.948, 214.412, 106.401, 43.836, 26.033]
  MoveL 3455 to (61.69, 14.21, -237.69) mm, rotated rx -152.51 ry -6.42 rz -112.51 deg; joints [10.771, -31.135, 88.079, 214.432, 106.518, 43.923, 26.033]
  MoveL 3456 to (62.21, 12.13, -237.89) mm, rotated rx -152.51 ry -6.42 rz -112.51 deg; joints [10.765, -31.129, 88.218, 214.452, 106.636, 44.012, 26.033]
  MoveL 3457 to (63.23, 7.99, -238.09) mm, rotated rx -152.51 ry -6.42 rz -112.51 deg; joints [10.754, -31.101, 88.476, 214.493, 106.868, 44.186, 26.033]
  MoveL 3458 to (63.65, 6.25, -238.3) mm, rotated rx -152.51 ry -6.42 rz -112.51 deg; joints [10.749, -31.097, 88.595, 214.51, 106.968, 44.261, 26.033]
  MoveL 3459 to (64.16, 4.35, -238.38) mm, rotated rx -152.51 ry -6.42 rz -112.51 deg; joints [10.742, -31.082, 88.711, 214.528, 107.073, 44.342, 26.033]
  MoveL 3460 to (64.74, 2.38, -238.39) mm, rotated rx -152.51 ry -6.42 rz -112.51 deg; joints [10.734, -31.061, 88.825, 214.546, 107.182, 44.426, 26.033]
  MoveL 3461 to (65.36, -0.22, -238.5) mm, rotated rx -152.51 ry -6.42 rz -112.51 deg; joints [10.727, -31.041, 88.983, 214.573, 107.327, 44.535, 26.033]
  MoveL 3462 to (65.85, -2.75, -238.59) mm, rotated rx -152.51 ry -6.42 rz -112.51 deg; joints [10.725, -31.021, 89.135, 214.602, 107.468, 44.638, 26.033]
  MoveL 3463 to (66.33, -4.91, -238.69) mm, rotated rx -152.51 ry -6.42 rz -112.51 deg; joints [10.721, -31.004, 89.266, 214.626, 107.589, 44.728, 26.033]
  MoveL 3464 to (66.79, -6.9, -238.86) mm, rotated rx -152.51 ry -6.42 rz -112.51 deg; joints [10.716, -30.994, 89.394, 214.647, 107.701, 44.813, 26.033]
  MoveL 3465 to (67.21, -8.76, -239.14) mm, rotated rx -152.51 ry -6.42 rz -112.51 deg; joints [10.711, -30.992, 89.524, 214.668, 107.808, 44.894, 26.033]
  MoveL 3466 to (67.62, -10.61, -239.43) mm, rotated rx -152.51 ry -6.42 rz -112.51 deg; joints [10.707, -30.99, 89.654, 214.688, 107.915, 44.974, 26.033]
  MoveL 3467 to (68, -12.45, -239.72) mm, rotated rx -152.51 ry -6.42 rz -112.51 deg; joints [10.703, -30.989, 89.783, 214.71, 108.021, 45.054, 26.033]
  MoveL 3468 to (68.43, -14.39, -239.87) mm, rotated rx -152.51 ry -6.42 rz -112.51 deg; joints [10.699, -30.977, 89.905, 214.732, 108.13, 45.136, 26.033]
  MoveL 3469 to (68.1, -14.95, -240.5) mm, rotated rx -152.51 ry -6.42 rz -112.51 deg; joints [10.711, -31.017, 89.994, 214.75, 108.174, 45.16, 26.033]
  MoveL 3470 to (67.89, -14.71, -240.8) mm, rotated rx -152.51 ry -6.42 rz -112.51 deg; joints [10.715, -31.042, 90.008, 214.751, 108.166, 45.152, 26.033]
  MoveL 3471 to (67.85, -14.71, -241) mm, rotated rx -152.51 ry -6.42 rz -112.51 deg; joints [10.716, -31.056, 90.026, 214.752, 108.17, 45.154, 26.033]
  MoveL 3472 to (67.96, -14.94, -241.09) mm, rotated rx -152.51 ry -6.42 rz -112.51 deg; joints [10.713, -31.059, 90.047, 214.753, 108.184, 45.166, 26.033]
  MoveL 3473 to (68.22, -15.3, -241.11) mm, rotated rx -152.51 ry -6.42 rz -112.51 deg; joints [10.706, -31.054, 90.068, 214.753, 108.203, 45.185, 26.033]
  MoveL 3474 to (68.54, -15.67, -241.12) mm, rotated rx -152.51 ry -6.42 rz -112.51 deg; joints [10.697, -31.047, 90.088, 214.752, 108.222, 45.205, 26.033]
  MoveL 3475 to (69.26, -16.33, -241.15) mm, rotated rx -152.51 ry -6.42 rz -112.51 deg; joints [10.676, -31.035, 90.126, 214.746, 108.257, 45.244, 26.033]
  MoveL 3476 to (70.42, -17.39, -241.15) mm, rotated rx -152.51 ry -6.42 rz -112.51 deg; joints [10.642, -31.012, 90.182, 214.737, 108.312, 45.307, 26.033]
  MoveL 3477 to (71.12, -18.08, -241.17) mm, rotated rx -152.51 ry -6.42 rz -112.51 deg; joints [10.622, -30.998, 90.219, 214.732, 108.348, 45.346, 26.033]
  MoveL 3478 to (71.89, -18.78, -241.17) mm, rotated rx -152.51 ry -6.42 rz -112.51 deg; joints [10.6, -30.983, 90.256, 214.725, 108.385, 45.387, 26.033]
  MoveL 3479 to (72.27, -19.14, -241.18) mm, rotated rx -152.51 ry -6.42 rz -112.51 deg; joints [10.589, -30.976, 90.276, 214.723, 108.403, 45.408, 26.033]
  MoveL 3480 to (72.61, -19.47, -241.21) mm, rotated rx -152.51 ry -6.42 rz -112.51 deg; joints [10.579, -30.971, 90.296, 214.72, 108.421, 45.427, 26.033]
  MoveL 3481 to (72.92, -19.78, -241.26) mm, rotated rx -152.51 ry -6.42 rz -112.51 deg; joints [10.57, -30.968, 90.316, 214.718, 108.438, 45.446, 26.033]
  MoveL 3482 to (73.19, -20.07, -241.32) mm, rotated rx -152.51 ry -6.42 rz -112.51 deg; joints [10.562, -30.966, 90.337, 214.717, 108.454, 45.463, 26.033]
  MoveL 3483 to (73.49, -20.37, -241.37) mm, rotated rx -152.51 ry -6.42 rz -112.51 deg; joints [10.553, -30.963, 90.358, 214.715, 108.471, 45.481, 26.033]
  MoveL 3484 to (73.82, -20.7, -241.41) mm, rotated rx -152.51 ry -6.42 rz -112.51 deg; joints [10.544, -30.959, 90.378, 214.713, 108.488, 45.5, 26.033]
  MoveL 3485 to (74.16, -21.03, -241.43) mm, rotated rx -152.51 ry -6.42 rz -112.51 deg; joints [10.534, -30.953, 90.397, 214.71, 108.506, 45.519, 26.033]
  MoveL 3486 to (74.46, -21.34, -241.47) mm, rotated rx -152.51 ry -6.42 rz -112.51 deg; joints [10.525, -30.949, 90.418, 214.708, 108.523, 45.537, 26.033]
  MoveL 3487 to (74.73, -21.65, -241.53) mm, rotated rx -152.51 ry -6.42 rz -112.51 deg; joints [10.517, -30.947, 90.439, 214.707, 108.54, 45.555, 26.033]
  MoveL 3488 to (75.01, -21.95, -241.58) mm, rotated rx -152.51 ry -6.42 rz -112.51 deg; joints [10.509, -30.945, 90.459, 214.706, 108.556, 45.572, 26.033]
  MoveL 3489 to (75.32, -22.26, -241.62) mm, rotated rx -152.51 ry -6.42 rz -112.51 deg; joints [10.5, -30.94, 90.478, 214.704, 108.573, 45.59, 26.033]
  MoveL 3490 to (75.7, -22.61, -241.62) mm, rotated rx -152.51 ry -6.42 rz -112.51 deg; joints [10.489, -30.932, 90.496, 214.701, 108.592, 45.611, 26.033]
  MoveL 3491 to (77.68, -24.76, -241.97) mm, rotated rx -152.51 ry -6.42 rz -112.51 deg; joints [10.431, -30.912, 90.64, 214.691, 108.71, 45.735, 26.033]
  MoveL 3492 to (78.39, -25.84, -242.42) mm, rotated rx -152.51 ry -6.42 rz -112.51 deg; joints [10.411, -30.922, 90.737, 214.692, 108.775, 45.795, 26.033]
  MoveL 3493 to (78.91, -26.92, -243.04) mm, rotated rx -152.51 ry -6.42 rz -112.51 deg; joints [10.396, -30.947, 90.85, 214.699, 108.844, 45.855, 26.033]
  MoveL 3494 to (79.4, -29.08, -244.82) mm, rotated rx -152.51 ry -6.42 rz -112.51 deg; joints [10.382, -31.037, 91.126, 214.725, 108.993, 45.973, 26.033]
  MoveL 3495 to (79.15, -31.26, -247.31) mm, rotated rx -152.51 ry -6.42 rz -112.51 deg; joints [10.391, -31.182, 91.468, 214.771, 109.157, 46.088, 26.033]
  MoveL 3496 to (78.34, -32.86, -249.81) mm, rotated rx -152.51 ry -6.42 rz -112.51 deg; joints [10.416, -31.34, 91.78, 214.819, 109.291, 46.171, 26.033]
  MoveL 3497 to (77.8, -33.24, -250.79) mm, rotated rx -152.51 ry -6.42 rz -112.51 deg; joints [10.432, -31.407, 91.889, 214.839, 109.33, 46.19, 26.033]
  MoveL 3498 to (77.17, -33.33, -251.59) mm, rotated rx -152.51 ry -6.42 rz -112.51 deg; joints [10.45, -31.466, 91.967, 214.856, 109.35, 46.193, 26.033]
  MoveL 3499 to (76.82, -33.27, -251.92) mm, rotated rx -152.51 ry -6.42 rz -112.51 deg; joints [10.46, -31.493, 91.995, 214.864, 109.354, 46.189, 26.033]
  MoveL 3500 to (76.45, -33.13, -252.21) mm, rotated rx -152.51 ry -6.42 rz -112.51 deg; joints [10.471, -31.518, 92.014, 214.871, 109.352, 46.181, 26.033]
  MoveL 3501 to (75.63, -32.65, -252.66) mm, rotated rx -152.51 ry -6.42 rz -112.51 deg; joints [10.494, -31.562, 92.031, 214.882, 109.336, 46.154, 26.033]
  MoveL 3502 to (74.73, -31.88, -252.92) mm, rotated rx -152.51 ry -6.42 rz -112.51 deg; joints [10.52, -31.598, 92.016, 214.89, 109.301, 46.112, 26.033]
  MoveL 3503 to (73.73, -30.83, -253.01) mm, rotated rx -152.51 ry -6.42 rz -112.51 deg; joints [10.548, -31.627, 91.969, 214.896, 109.247, 46.055, 26.033]
  MoveL 3504 to (72.01, -28.85, -253.01) mm, rotated rx -152.51 ry -6.42 rz -112.51 deg; joints [10.596, -31.668, 91.867, 214.902, 109.144, 45.947, 26.033]
  MoveL 3505 to (71.73, -28.51, -252.98) mm, rotated rx -152.51 ry -6.42 rz -112.51 deg; joints [10.604, -31.673, 91.847, 214.903, 109.125, 45.929, 26.033]
  MoveL 3506 to (71.49, -28.19, -252.93) mm, rotated rx -152.51 ry -6.42 rz -112.51 deg; joints [10.611, -31.676, 91.826, 214.903, 109.108, 45.911, 26.033]
  MoveL 3507 to (71.26, -27.88, -252.87) mm, rotated rx -152.51 ry -6.42 rz -112.51 deg; joints [10.617, -31.677, 91.803, 214.903, 109.09, 45.894, 26.033]
  MoveL 3508 to (71, -27.54, -252.82) mm, rotated rx -152.51 ry -6.42 rz -112.51 deg; joints [10.624, -31.68, 91.781, 214.903, 109.071, 45.875, 26.033]
  MoveL 3509 to (70.68, -27.15, -252.78) mm, rotated rx -152.51 ry -6.42 rz -112.51 deg; joints [10.633, -31.685, 91.757, 214.904, 109.05, 45.854, 26.033]
  MoveL 3510 to (70.36, -26.74, -252.72) mm, rotated rx -152.51 ry -6.42 rz -112.51 deg; joints [10.642, -31.69, 91.731, 214.904, 109.027, 45.832, 26.033]
  MoveL 3511 to (70.01, -26.32, -252.7) mm, rotated rx -152.51 ry -6.42 rz -112.51 deg; joints [10.652, -31.697, 91.707, 214.905, 109.005, 45.809, 26.033]
  MoveL 3512 to (69.59, -25.84, -252.72) mm, rotated rx -152.51 ry -6.42 rz -112.51 deg; joints [10.664, -31.708, 91.683, 214.907, 108.98, 45.783, 26.033]
  MoveL 3513 to (69, -25.2, -252.78) mm, rotated rx -152.51 ry -6.42 rz -112.51 deg; joints [10.68, -31.725, 91.656, 214.91, 108.948, 45.748, 26.033]
  MoveL 3514 to (68.65, -24.81, -252.78) mm, rotated rx -152.51 ry -6.42 rz -112.51 deg; joints [10.69, -31.733, 91.635, 214.911, 108.927, 45.727, 26.033]
  MoveL 3515 to (68.33, -24.43, -252.78) mm, rotated rx -152.51 ry -6.42 rz -112.51 deg; joints [10.699, -31.74, 91.615, 214.913, 108.907, 45.706, 26.033]
  MoveL 3516 to (68.03, -24.07, -252.76) mm, rotated rx -152.51 ry -6.42 rz -112.51 deg; joints [10.707, -31.746, 91.594, 214.914, 108.888, 45.687, 26.033]
  MoveL 3517 to (67.78, -23.74, -252.7) mm, rotated rx -152.51 ry -6.42 rz -112.51 deg; joints [10.714, -31.749, 91.572, 214.914, 108.869, 45.669, 26.033]
  MoveL 3518 to (67.55, -23.41, -252.65) mm, rotated rx -152.51 ry -6.42 rz -112.51 deg; joints [10.72, -31.751, 91.55, 214.913, 108.851, 45.651, 26.033]
  MoveL 3519 to (67.35, -23.04, -252.6) mm, rotated rx -152.51 ry -6.42 rz -112.51 deg; joints [10.725, -31.754, 91.525, 214.912, 108.83, 45.633, 26.033]
  MoveL 3520 to (67.19, -22.66, -252.54) mm, rotated rx -152.51 ry -6.42 rz -112.51 deg; joints [10.729, -31.755, 91.5, 214.909, 108.809, 45.614, 26.033]
  MoveL 3521 to (67.16, -22.44, -252.38) mm, rotated rx -152.51 ry -6.42 rz -112.51 deg; joints [10.729, -31.747, 91.473, 214.906, 108.794, 45.603, 26.033]
  MoveL 3522 to (67.26, -22.49, -252.06) mm, rotated rx -152.51 ry -6.42 rz -112.51 deg; joints [10.728, -31.725, 91.448, 214.904, 108.791, 45.602, 26.033]
  MoveL 3523 to (67.49, -22.86, -251.57) mm, rotated rx -152.51 ry -6.42 rz -112.51 deg; joints [10.724, -31.686, 91.424, 214.905, 108.803, 45.613, 26.033]
  MoveL 3524 to (67.35, -21.99, -250.72) mm, rotated rx -152.51 ry -6.42 rz -112.51 deg; joints [10.728, -31.639, 91.301, 214.892, 108.74, 45.564, 26.033]
  MoveL 3525 to (66.81, -17.75, -250.72) mm, rotated rx -152.51 ry -6.42 rz -112.51 deg; joints [10.722, -31.687, 91.067, 214.833, 108.507, 45.397, 26.033]
  MoveL 3526 to (66.56, -15.77, -250.65) mm, rotated rx -152.51 ry -6.42 rz -112.51 deg; joints [10.719, -31.705, 90.95, 214.806, 108.397, 45.318, 26.033]
  MoveL 3527 to (66.33, -13.79, -250.51) mm, rotated rx -152.51 ry -6.42 rz -112.51 deg; joints [10.716, -31.716, 90.827, 214.778, 108.285, 45.238, 26.033]
  MoveL 3528 to (66.06, -11.51, -250.31) mm, rotated rx -152.51 ry -6.42 rz -112.51 deg; joints [10.712, -31.727, 90.682, 214.746, 108.156, 45.146, 26.033]
  MoveL 3529 to (65.81, -9.35, -250.1) mm, rotated rx -152.51 ry -6.42 rz -112.51 deg; joints [10.709, -31.736, 90.542, 214.717, 108.033, 45.059, 26.033]
  MoveL 3530 to (65.54, -7.19, -249.99) mm, rotated rx -152.51 ry -6.42 rz -112.51 deg; joints [10.706, -31.751, 90.411, 214.687, 107.911, 44.972, 26.033]
  MoveL 3531 to (65.27, -5.07, -249.99) mm, rotated rx -152.51 ry -6.42 rz -112.51 deg; joints [10.703, -31.773, 90.291, 214.659, 107.794, 44.889, 26.033]
  MoveL 3532 to (65.02, -3.1, -249.93) mm, rotated rx -152.51 ry -6.42 rz -112.51 deg; joints [10.7, -31.788, 90.174, 214.633, 107.684, 44.811, 26.033]
  MoveL 3533 to (64.77, -1.24, -249.81) mm, rotated rx -152.51 ry -6.42 rz -112.51 deg; joints [10.698, -31.799, 90.057, 214.608, 107.579, 44.736, 26.033]
  MoveL 3534 to (64.51, 0.78, -249.75) mm, rotated rx -152.51 ry -6.42 rz -112.51 deg; joints [10.695, -31.814, 89.936, 214.582, 107.465, 44.656, 26.033]
  MoveL 3535 to (64.24, 2.9, -249.56) mm, rotated rx -152.51 ry -6.42 rz -112.51 deg; joints [10.693, -31.822, 89.798, 214.554, 107.345, 44.571, 26.033]
  MoveL 3536 to (63.7, 7.13, -249.38) mm, rotated rx -152.51 ry -6.42 rz -112.51 deg; joints [10.687, -31.85, 89.538, 214.5, 107.106, 44.403, 26.033]
  MoveL 3537 to (63.42, 9.25, -249.2) mm, rotated rx -152.51 ry -6.42 rz -112.51 deg; joints [10.686, -31.857, 89.4, 214.473, 106.986, 44.317, 26.033]
  MoveL 3538 to (63.13, 11.36, -249.02) mm, rotated rx -152.51 ry -6.42 rz -112.51 deg; joints [10.684, -31.864, 89.261, 214.447, 106.865, 44.232, 26.033]
  MoveL 3539 to (62.86, 13.48, -249.02) mm, rotated rx -152.51 ry -6.42 rz -112.51 deg; joints [10.68, -31.883, 89.137, 214.42, 106.747, 44.149, 26.033]
  MoveL 3540 to (62.57, 15.6, -248.85) mm, rotated rx -152.51 ry -6.42 rz -112.51 deg; joints [10.679, -31.889, 88.998, 214.394, 106.626, 44.064, 26.033]
  MoveL 3541 to (62.27, 17.71, -248.67) mm, rotated rx -152.51 ry -6.42 rz -112.51 deg; joints [10.677, -31.895, 88.858, 214.369, 106.505, 43.979, 26.033]
  MoveL 3542 to (62, 19.83, -248.67) mm, rotated rx -152.51 ry -6.42 rz -112.51 deg; joints [10.674, -31.913, 88.733, 214.343, 106.386, 43.896, 26.033]
  MoveL 3543 to (61.68, 21.75, -248.47) mm, rotated rx -152.51 ry -6.42 rz -112.51 deg; joints [10.675, -31.916, 88.602, 214.321, 106.276, 43.817, 26.033]
  MoveL 3544 to (61.34, 23.43, -248.15) mm, rotated rx -152.51 ry -6.42 rz -112.51 deg; joints [10.678, -31.909, 88.474, 214.304, 106.177, 43.745, 26.033]
  MoveL 3545 to (60.95, 24.91, -247.69) mm, rotated rx -152.51 ry -6.42 rz -112.51 deg; joints [10.685, -31.891, 88.345, 214.29, 106.087, 43.676, 26.033]
  MoveL 3546 to (60.9, 23.96, -246.92) mm, rotated rx -152.51 ry -6.42 rz -112.51 deg; joints [10.696, -31.834, 88.333, 214.305, 106.128, 43.698, 26.033]
  MoveL 3547 to (60.89, 24.37, -246.92) mm, rotated rx -152.51 ry -6.42 rz -112.51 deg; joints [10.694, -31.836, 88.308, 214.299, 106.105, 43.682, 26.033]
  MoveC 3548 to (62.22, 27.67, -246.92) mm, rotated rx -152.51 ry -6.42 rz -112.51 deg; joints [10.629, -31.842, 88.107, 214.221, 105.913, 43.592, 26.033] to (63.82, 30.85, -246.92) mm, rotated rx -152.51 ry -6.42 rz -112.51 deg; joints [10.557, -31.844, 87.911, 214.139, 105.727, 43.511, 26.033]
  MoveL 3549 to (63.82, 30.85, -246.92) mm, rotated rx -152.51 ry -6.42 rz -112.51 deg; joints [10.557, -31.844, 87.911, 214.139, 105.727, 43.511, 26.033]
  MoveL 3550 to (64.02, 31.27, -246.89) mm, rotated rx -152.51 ry -6.42 rz -112.51 deg; joints [10.548, -31.843, 87.883, 214.128, 105.702, 43.5, 26.033]
  MoveL 3551 to (64.18, 31.66, -246.84) mm, rotated rx -152.51 ry -6.42 rz -112.51 deg; joints [10.54, -31.84, 87.854, 214.119, 105.678, 43.488, 26.033]
  MoveL 3552 to (64.33, 32.04, -246.78) mm, rotated rx -152.51 ry -6.42 rz -112.51 deg; joints [10.533, -31.836, 87.825, 214.11, 105.655, 43.477, 26.033]
  MoveL 3553 to (64.51, 32.44, -246.74) mm, rotated rx -152.51 ry -6.42 rz -112.51 deg; joints [10.525, -31.833, 87.796, 214.1, 105.631, 43.466, 26.033]
  MoveL 3554 to (64.7, 32.87, -246.71) mm, rotated rx -152.51 ry -6.42 rz -112.51 deg; joints [10.516, -31.832, 87.767, 214.089, 105.605, 43.454, 26.033]
  MoveL 3555 to (64.93, 33.34, -246.69) mm, rotated rx -152.51 ry -6.42 rz -112.51 deg; joints [10.506, -31.831, 87.737, 214.078, 105.577, 43.442, 26.033]
  MoveL 3556 to (65.4, 34.27, -246.69) mm, rotated rx -152.51 ry -6.42 rz -112.51 deg; joints [10.485, -31.831, 87.679, 214.054, 105.522, 43.418, 26.033]
  MoveL 3557 to (66.1, 35.55, -246.79) mm, rotated rx -152.51 ry -6.42 rz -112.51 deg; joints [10.453, -31.837, 87.607, 214.02, 105.449, 43.388, 26.033]
  MoveL 3558 to (66.78, 36.54, -247.06) mm, rotated rx -152.51 ry -6.42 rz -112.51 deg; joints [10.423, -31.853, 87.57, 213.99, 105.394, 43.372, 26.033]
  MoveL 3559 to (67.45, 37.23, -247.52) mm, rotated rx -152.51 ry -6.42 rz -112.51 deg; joints [10.394, -31.881, 87.566, 213.965, 105.36, 43.368, 26.033]
  MoveL 3560 to (68.11, 37.64, -248.16) mm, rotated rx -152.51 ry -6.42 rz -112.51 deg; joints [10.366, -31.919, 87.597, 213.945, 105.344, 43.377, 26.033]
  MoveL 3561 to (68.74, 37.76, -248.98) mm, rotated rx -152.51 ry -6.42 rz -112.51 deg; joints [10.34, -31.969, 87.662, 213.929, 105.349, 43.398, 26.033]
  MoveL 3562 to (69.36, 37.6, -249.98) mm, rotated rx -152.51 ry -6.42 rz -112.51 deg; joints [10.315, -32.03, 87.76, 213.917, 105.372, 43.432, 26.033]
  MoveL 3563 to (70.55, 36.39, -252.54) mm, rotated rx -152.51 ry -6.42 rz -112.51 deg; joints [10.269, -32.183, 88.059, 213.907, 105.478, 43.539, 26.033]
  MoveL 3564 to (71.35, 34.5, -255.1) mm, rotated rx -152.51 ry -6.42 rz -112.51 deg; joints [10.239, -32.337, 88.4, 213.916, 105.624, 43.661, 26.033]
  MoveL 3565 to (71.48, 33.48, -256.11) mm, rotated rx -152.51 ry -6.42 rz -112.51 deg; joints [10.236, -32.398, 88.551, 213.927, 105.698, 43.715, 26.033]
  MoveL 3566 to (71.43, 32.39, -256.93) mm, rotated rx -152.51 ry -6.42 rz -112.51 deg; joints [10.239, -32.447, 88.69, 213.944, 105.773, 43.765, 26.033]
  MoveL 3567 to (71.2, 31.25, -257.57) mm, rotated rx -152.51 ry -6.42 rz -112.51 deg; joints [10.25, -32.486, 88.816, 213.965, 105.849, 43.811, 26.033]
  MoveL 3568 to (70.79, 30.06, -258.03) mm, rotated rx -152.51 ry -6.42 rz -112.51 deg; joints [10.269, -32.514, 88.93, 213.992, 105.926, 43.852, 26.033]
  MoveL 3569 to (69.43, 27.5, -258.4) mm, rotated rx -152.51 ry -6.42 rz -112.51 deg; joints [10.328, -32.538, 89.12, 214.06, 106.082, 43.921, 26.033]
  MoveL 3570 to (68.86, 26.62, -258.4) mm, rotated rx -152.51 ry -6.42 rz -112.51 deg; joints [10.352, -32.538, 89.175, 214.086, 106.135, 43.94, 26.033]
  MoveL 3571 to (68.58, 26.18, -258.4) mm, rotated rx -152.51 ry -6.42 rz -112.51 deg; joints [10.365, -32.539, 89.203, 214.099, 106.161, 43.951, 26.033]
  MoveL 3572 to (68.33, 25.77, -258.43) mm, rotated rx -152.51 ry -6.42 rz -112.51 deg; joints [10.375, -32.541, 89.23, 214.111, 106.185, 43.96, 26.033]
  MoveL 3573 to (68.13, 25.4, -258.48) mm, rotated rx -152.51 ry -6.42 rz -112.51 deg; joints [10.384, -32.544, 89.257, 214.121, 106.208, 43.97, 26.033]
  MoveL 3574 to (67.93, 25.04, -258.53) mm, rotated rx -152.51 ry -6.42 rz -112.51 deg; joints [10.392, -32.547, 89.283, 214.131, 106.229, 43.98, 26.033]
  MoveL 3575 to (67.73, 24.68, -258.58) mm, rotated rx -152.51 ry -6.42 rz -112.51 deg; joints [10.401, -32.551, 89.31, 214.141, 106.252, 43.989, 26.033]
  MoveL 3576 to (67.49, 24.28, -258.6) mm, rotated rx -152.51 ry -6.42 rz -112.51 deg; joints [10.412, -32.552, 89.336, 214.152, 106.276, 43.999, 26.033]
  MoveL 3577 to (67.22, 23.86, -258.61) mm, rotated rx -152.51 ry -6.42 rz -112.51 deg; joints [10.423, -32.553, 89.363, 214.165, 106.301, 44.009, 26.033]
  MoveL 3578 to (66.92, 23.39, -258.6) mm, rotated rx -152.51 ry -6.42 rz -112.51 deg; joints [10.436, -32.552, 89.391, 214.178, 106.328, 44.019, 26.033]
  MoveL 3579 to (66.63, 22.95, -258.61) mm, rotated rx -152.51 ry -6.42 rz -112.51 deg; joints [10.449, -32.553, 89.419, 214.192, 106.354, 44.029, 26.033]
  MoveL 3580 to (66.37, 22.53, -258.63) mm, rotated rx -152.51 ry -6.42 rz -112.51 deg; joints [10.46, -32.555, 89.447, 214.204, 106.38, 44.04, 26.033]
  MoveL 3581 to (66.13, 22.12, -258.68) mm, rotated rx -152.51 ry -6.42 rz -112.51 deg; joints [10.47, -32.558, 89.476, 214.215, 106.404, 44.05, 26.033]
  MoveL 3582 to (65.89, 21.67, -258.75) mm, rotated rx -152.51 ry -6.42 rz -112.51 deg; joints [10.481, -32.562, 89.51, 214.228, 106.432, 44.062, 26.033]
  MoveL 3583 to (65.6, 21.14, -258.82) mm, rotated rx -152.51 ry -6.42 rz -112.51 deg; joints [10.493, -32.566, 89.548, 214.242, 106.464, 44.076, 26.033]
  MoveL 3584 to (65.3, 20.66, -258.83) mm, rotated rx -152.51 ry -6.42 rz -112.51 deg; joints [10.506, -32.567, 89.579, 214.256, 106.492, 44.088, 26.033]
  MoveL 3585 to (65.02, 20.21, -258.84) mm, rotated rx -152.51 ry -6.42 rz -112.51 deg; joints [10.519, -32.567, 89.606, 214.27, 106.519, 44.098, 26.033]
  MoveL 3586 to (64.73, 19.77, -258.84) mm, rotated rx -152.51 ry -6.42 rz -112.51 deg; joints [10.531, -32.568, 89.633, 214.283, 106.545, 44.108, 26.033]
  MoveL 3587 to (64.39, 19.21, -258.85) mm, rotated rx -152.51 ry -6.42 rz -112.51 deg; joints [10.546, -32.568, 89.668, 214.299, 106.578, 44.121, 26.033]
  MoveL 3588 to (64.11, 18.7, -258.86) mm, rotated rx -152.51 ry -6.42 rz -112.51 deg; joints [10.558, -32.568, 89.7, 214.313, 106.608, 44.134, 26.033]
  MoveL 3589 to (63.89, 18.24, -258.86) mm, rotated rx -152.51 ry -6.42 rz -112.51 deg; joints [10.569, -32.568, 89.728, 214.325, 106.634, 44.146, 26.033]
  MoveL 3590 to (63.79, 17.92, -258.87) mm, rotated rx -152.51 ry -6.42 rz -112.51 deg; joints [10.574, -32.567, 89.748, 214.333, 106.653, 44.156, 26.033]
  MoveL 3591 to (63.75, 17.65, -258.87) mm, rotated rx -152.51 ry -6.42 rz -112.51 deg; joints [10.577, -32.565, 89.764, 214.338, 106.669, 44.165, 26.033]
  MoveL 3592 to (63.86, 18.58, -259.46) mm, rotated rx -152.51 ry -6.42 rz -112.51 deg; joints [10.565, -32.61, 89.761, 214.321, 106.625, 44.142, 26.033]
  MoveL 3593 to (64.16, 17.28, -259.99) mm, rotated rx -152.51 ry -6.42 rz -112.51 deg; joints [10.559, -32.633, 89.883, 214.334, 106.706, 44.203, 26.033]
  MoveL 3594 to (64.37, 15.73, -260.37) mm, rotated rx -152.51 ry -6.42 rz -112.51 deg; joints [10.559, -32.645, 90.008, 214.353, 106.798, 44.269, 26.033]
  MoveL 3595 to (64.5, 13.89, -260.63) mm, rotated rx -152.51 ry -6.42 rz -112.51 deg; joints [10.564, -32.648, 90.138, 214.378, 106.906, 44.342, 26.033]
  MoveL 3596 to (64.57, 11.83, -260.75) mm, rotated rx -152.51 ry -6.42 rz -112.51 deg; joints [10.573, -32.64, 90.269, 214.409, 107.023, 44.42, 26.033]
  MoveL 3597 to (64.62, 9.73, -260.84) mm, rotated rx -152.51 ry -6.42 rz -112.51 deg; joints [10.583, -32.629, 90.4, 214.44, 107.143, 44.499, 26.033]
  MoveL 3598 to (64.72, 5.47, -261.02) mm, rotated rx -152.51 ry -6.42 rz -112.51 deg; joints [10.604, -32.606, 90.663, 214.506, 107.385, 44.659, 26.033]
  MoveL 3599 to (64.78, 3.33, -261.2) mm, rotated rx -152.51 ry -6.42 rz -112.51 deg; joints [10.614, -32.6, 90.801, 214.538, 107.507, 44.741, 26.033]
  MoveL 3600 to (64.86, -0.93, -261.38) mm, rotated rx -152.51 ry -6.42 rz -112.51 deg; joints [10.636, -32.575, 91.062, 214.605, 107.749, 44.901, 26.033]
  MoveL 3601 to (64.91, -3.06, -261.57) mm, rotated rx -152.51 ry -6.42 rz -112.51 deg; joints [10.646, -32.568, 91.2, 214.639, 107.871, 44.983, 26.033]
  MoveL 3602 to (64.95, -5.2, -261.66) mm, rotated rx -152.51 ry -6.42 rz -112.51 deg; joints [10.657, -32.554, 91.329, 214.673, 107.991, 45.063, 26.033]
  MoveL 3603 to (64.96, -7.17, -261.87) mm, rotated rx -152.51 ry -6.42 rz -112.51 deg; joints [10.667, -32.55, 91.46, 214.705, 108.105, 45.139, 26.033]
  MoveL 3604 to (65.01, -9.53, -262.02) mm, rotated rx -152.51 ry -6.42 rz -112.51 deg; joints [10.679, -32.538, 91.606, 214.743, 108.239, 45.229, 26.033]
  MoveL 3605 to (65.05, -12.09, -262.13) mm, rotated rx -152.51 ry -6.42 rz -112.51 deg; joints [10.692, -32.521, 91.76, 214.785, 108.384, 45.326, 26.033]
  MoveL 3606 to (65.09, -14.23, -262.13) mm, rotated rx -152.51 ry -6.42 rz -112.51 deg; joints [10.703, -32.5, 91.88, 214.82, 108.502, 45.406, 26.033]
  MoveL 3607 to (65.12, -16.26, -262.21) mm, rotated rx -152.51 ry -6.42 rz -112.51 deg; joints [10.714, -32.485, 92, 214.854, 108.617, 45.483, 26.033]
  MoveL 3608 to (65.13, -18.09, -262.38) mm, rotated rx -152.51 ry -6.42 rz -112.51 deg; joints [10.724, -32.478, 92.118, 214.885, 108.721, 45.553, 26.033]
  MoveL 3609 to (65.13, -19.96, -262.59) mm, rotated rx -152.51 ry -6.42 rz -112.51 deg; joints [10.734, -32.473, 92.24, 214.917, 108.828, 45.625, 26.033]
  MoveL 3610 to (65.16, -22.32, -262.73) mm, rotated rx -152.51 ry -6.42 rz -112.51 deg; joints [10.747, -32.458, 92.383, 214.957, 108.962, 45.716, 26.033]
  MoveL 3611 to (65.19, -24.9, -262.84) mm, rotated rx -152.51 ry -6.42 rz -112.51 deg; joints [10.761, -32.438, 92.534, 215.001, 109.106, 45.814, 26.033]
  MoveL 3612 to (65.27, -29.16, -262.84) mm, rotated rx -152.51 ry -6.42 rz -112.51 deg; joints [10.784, -32.392, 92.768, 215.074, 109.342, 45.974, 26.033]
  MoveL 3613 to (65.04, -29.38, -263.53) mm, rotated rx -152.51 ry -6.42 rz -112.51 deg; joints [10.79, -32.438, 92.841, 215.084, 109.366, 45.988, 26.033]
  MoveL 3614 to (64.91, -29.09, -263.88) mm, rotated rx -152.51 ry -6.42 rz -112.51 deg; joints [10.791, -32.465, 92.856, 215.082, 109.356, 45.98, 26.033]
  MoveL 3615 to (64.89, -29.09, -264.1) mm, rotated rx -152.51 ry -6.42 rz -112.51 deg; joints [10.79, -32.48, 92.875, 215.083, 109.359, 45.983, 26.033]
  MoveL 3616 to (64.98, -29.34, -264.21) mm, rotated rx -152.51 ry -6.42 rz -112.51 deg; joints [10.788, -32.483, 92.898, 215.085, 109.375, 45.996, 26.033]
  MoveL 3617 to (65.19, -29.74, -264.24) mm, rotated rx -152.51 ry -6.42 rz -112.51 deg; joints [10.783, -32.479, 92.922, 215.087, 109.397, 46.015, 26.033]
  MoveL 3618 to (65.44, -30.15, -264.26) mm, rotated rx -152.51 ry -6.42 rz -112.51 deg; joints [10.777, -32.473, 92.946, 215.089, 109.419, 46.036, 26.033]
  MoveL 3619 to (65.66, -30.52, -264.31) mm, rotated rx -152.51 ry -6.42 rz -112.51 deg; joints [10.771, -32.47, 92.97, 215.09, 109.44, 46.055, 26.033]
  MoveL 3620 to (65.86, -30.87, -264.38) mm, rotated rx -152.51 ry -6.42 rz -112.51 deg; joints [10.766, -32.468, 92.994, 215.091, 109.459, 46.073, 26.033]
  MoveL 3621 to (66.07, -31.22, -264.44) mm, rotated rx -152.51 ry -6.42 rz -112.51 deg; joints [10.76, -32.466, 93.017, 215.092, 109.479, 46.091, 26.033]
  MoveL 3622 to (66.31, -31.6, -264.48) mm, rotated rx -152.51 ry -6.42 rz -112.51 deg; joints [10.754, -32.462, 93.04, 215.093, 109.5, 46.11, 26.033]
  MoveL 3623 to (66.6, -32.03, -264.5) mm, rotated rx -152.51 ry -6.42 rz -112.51 deg; joints [10.746, -32.455, 93.065, 215.094, 109.523, 46.133, 26.033]
  MoveL 3624 to (66.88, -32.49, -264.56) mm, rotated rx -152.51 ry -6.42 rz -112.51 deg; joints [10.739, -32.451, 93.095, 215.096, 109.548, 46.156, 26.033]
  MoveL 3625 to (67.16, -32.92, -264.6) mm, rotated rx -152.51 ry -6.42 rz -112.51 deg; joints [10.731, -32.445, 93.12, 215.097, 109.572, 46.179, 26.033]
  MoveL 3626 to (67.46, -33.35, -264.6) mm, rotated rx -152.51 ry -6.42 rz -112.51 deg; joints [10.724, -32.437, 93.143, 215.097, 109.595, 46.201, 26.033]
  MoveL 3627 to (67.76, -33.78, -264.6) mm, rotated rx -152.51 ry -6.42 rz -112.51 deg; joints [10.716, -32.429, 93.166, 215.098, 109.618, 46.223, 26.033]
  MoveL 3628 to (68.17, -34.33, -264.57) mm, rotated rx -152.51 ry -6.42 rz -112.51 deg; joints [10.705, -32.416, 93.191, 215.098, 109.647, 46.251, 26.033]
  MoveL 3629 to (68.56, -34.87, -264.54) mm, rotated rx -152.51 ry -6.42 rz -112.51 deg; joints [10.695, -32.403, 93.217, 215.098, 109.675, 46.279, 26.033]
  MoveL 3630 to (68.9, -35.36, -264.53) mm, rotated rx -152.51 ry -6.42 rz -112.51 deg; joints [10.686, -32.393, 93.242, 215.099, 109.701, 46.304, 26.033]
  MoveL 3631 to (69.15, -35.76, -264.57) mm, rotated rx -152.51 ry -6.42 rz -112.51 deg; joints [10.679, -32.389, 93.265, 215.1, 109.722, 46.324, 26.033]
  MoveL 3632 to (69.37, -36.11, -264.63) mm, rotated rx -152.51 ry -6.42 rz -112.51 deg; joints [10.673, -32.386, 93.289, 215.101, 109.742, 46.343, 26.033]
  MoveL 3633 to (69.58, -36.46, -264.68) mm, rotated rx -152.51 ry -6.42 rz -112.51 deg; joints [10.668, -32.383, 93.312, 215.102, 109.762, 46.361, 26.033]
  MoveL 3634 to (69.81, -36.84, -264.72) mm, rotated rx -152.51 ry -6.42 rz -112.51 deg; joints [10.662, -32.378, 93.335, 215.103, 109.782, 46.38, 26.033]
  MoveL 3635 to (70.71, -38.12, -264.72) mm, rotated rx -152.51 ry -6.42 rz -112.51 deg; joints [10.638, -32.353, 93.401, 215.105, 109.851, 46.446, 26.033]
  MoveL 3636 to (72.17, -40.62, -265.09) mm, rotated rx -152.51 ry -6.42 rz -112.51 deg; joints [10.6, -32.332, 93.563, 215.115, 109.99, 46.574, 26.033]
  MoveL 3637 to (72.64, -41.78, -265.56) mm, rotated rx -152.51 ry -6.42 rz -112.51 deg; joints [10.588, -32.344, 93.665, 215.126, 110.06, 46.634, 26.033]
  MoveL 3638 to (72.92, -42.89, -266.22) mm, rotated rx -152.51 ry -6.42 rz -112.51 deg; joints [10.581, -32.371, 93.781, 215.139, 110.131, 46.691, 26.033]
  MoveL 3639 to (73.03, -43.94, -267.07) mm, rotated rx -152.51 ry -6.42 rz -112.51 deg; joints [10.579, -32.413, 93.91, 215.156, 110.202, 46.746, 26.033]
  MoveL 3640 to (72.96, -44.94, -268.11) mm, rotated rx -152.51 ry -6.42 rz -112.51 deg; joints [10.582, -32.469, 94.053, 215.177, 110.274, 46.797, 26.033]
  MoveL 3641 to (72.29, -46.77, -270.74) mm, rotated rx -152.51 ry -6.42 rz -112.51 deg; joints [10.604, -32.628, 94.381, 215.229, 110.418, 46.893, 26.033]
  MoveL 3642 to (71.2, -47.93, -273.38) mm, rotated rx -152.51 ry -6.42 rz -112.51 deg; joints [10.636, -32.799, 94.673, 215.279, 110.526, 46.954, 26.033]
  MoveL 3643 to (70.61, -48.08, -274.42) mm, rotated rx -152.51 ry -6.42 rz -112.51 deg; joints [10.652, -32.872, 94.773, 215.297, 110.552, 46.964, 26.033]
  MoveL 3644 to (69.98, -47.96, -275.26) mm, rotated rx -152.51 ry -6.42 rz -112.51 deg; joints [10.669, -32.936, 94.841, 215.31, 110.56, 46.959, 26.033]
  MoveL 3645 to (69.33, -47.55, -275.92) mm, rotated rx -152.51 ry -6.42 rz -112.51 deg; joints [10.687, -32.992, 94.878, 215.319, 110.549, 46.941, 26.033]
  MoveL 3646 to (68.64, -46.87, -276.39) mm, rotated rx -152.51 ry -6.42 rz -112.51 deg; joints [10.705, -33.039, 94.885, 215.323, 110.521, 46.908, 26.033]
  MoveL 3647 to (67.91, -45.9, -276.68) mm, rotated rx -152.51 ry -6.42 rz -112.51 deg; joints [10.723, -33.078, 94.86, 215.323, 110.474, 46.861, 26.033]
  MoveL 3648 to (67.16, -44.66, -276.77) mm, rotated rx -152.51 ry -6.42 rz -112.51 deg; joints [10.742, -33.108, 94.804, 215.318, 110.409, 46.8, 26.033]
  MoveL 3649 to (66.9, -44.2, -276.77) mm, rotated rx -152.51 ry -6.42 rz -112.51 deg; joints [10.748, -33.117, 94.78, 215.316, 110.384, 46.778, 26.033]
  MoveL 3650 to (66.69, -43.78, -276.75) mm, rotated rx -152.51 ry -6.42 rz -112.51 deg; joints [10.753, -33.123, 94.757, 215.314, 110.362, 46.758, 26.033]
  MoveL 3651 to (66.51, -43.42, -276.7) mm, rotated rx -152.51 ry -6.42 rz -112.51 deg; joints [10.757, -33.126, 94.734, 215.311, 110.341, 46.74, 26.033]
  MoveL 3652 to (66.35, -43.06, -276.65) mm, rotated rx -152.51 ry -6.42 rz -112.51 deg; joints [10.761, -33.129, 94.711, 215.308, 110.321, 46.722, 26.033]
  MoveL 3653 to (66.16, -42.68, -276.61) mm, rotated rx -152.51 ry -6.42 rz -112.51 deg; joints [10.766, -33.133, 94.687, 215.306, 110.3, 46.703, 26.033]
  MoveL 3654 to (65.94, -42.24, -276.58) mm, rotated rx -152.51 ry -6.42 rz -112.51 deg; joints [10.771, -33.139, 94.663, 215.303, 110.276, 46.682, 26.033]
  MoveL 3655 to (65.68, -41.78, -276.58) mm, rotated rx -152.51 ry -6.42 rz -112.51 deg; joints [10.777, -33.148, 94.639, 215.301, 110.251, 46.66, 26.033]
  MoveL 3656 to (65.46, -41.37, -276.56) mm, rotated rx -152.51 ry -6.42 rz -112.51 deg; joints [10.783, -33.154, 94.616, 215.298, 110.229, 46.639, 26.033]
  MoveL 3657 to (65.28, -41.01, -276.51) mm, rotated rx -152.51 ry -6.42 rz -112.51 deg; joints [10.787, -33.157, 94.592, 215.296, 110.209, 46.621, 26.033]
  MoveL 3658 to (65.11, -40.66, -276.44) mm, rotated rx -152.51 ry -6.42 rz -112.51 deg; joints [10.791, -33.159, 94.569, 215.294, 110.189, 46.604, 26.033]
  MoveL 3659 to (64.91, -40.27, -276.4) mm, rotated rx -152.51 ry -6.42 rz -112.51 deg; joints [10.796, -33.163, 94.545, 215.291, 110.168, 46.585, 26.033]
  MoveL 3660 to (64.68, -39.84, -276.37) mm, rotated rx -152.51 ry -6.42 rz -112.51 deg; joints [10.802, -33.169, 94.52, 215.289, 110.144, 46.563, 26.033]
  MoveL 3661 to (64.43, -39.38, -276.37) mm, rotated rx -152.51 ry -6.42 rz -112.51 deg; joints [10.808, -33.177, 94.496, 215.287, 110.119, 46.541, 26.033]
  MoveL 3662 to (64.01, -38.49, -276.35) mm, rotated rx -152.51 ry -6.42 rz -112.51 deg; joints [10.817, -33.191, 94.447, 215.28, 110.071, 46.498, 26.033]
  MoveC 3663 to (63.47, -37.22, -276.35) mm, rotated rx -152.51 ry -6.42 rz -112.51 deg; joints [10.829, -33.212, 94.381, 215.27, 110.002, 46.44, 26.033] to (62.77, -36.03, -276.35) mm, rotated rx -152.51 ry -6.42 rz -112.51 deg; joints [10.846, -33.234, 94.319, 215.265, 109.939, 46.381, 26.033]
  MoveL 3664 to (62.77, -36.03, -276.34) mm, rotated rx -152.51 ry -6.42 rz -112.51 deg; joints [10.846, -33.234, 94.318, 215.265, 109.938, 46.381, 26.033]
  MoveL 3665 to (62.49, -35.43, -276.33) mm, rotated rx -152.51 ry -6.42 rz -112.51 deg; joints [10.852, -33.243, 94.285, 215.261, 109.906, 46.352, 26.033]
  MoveL 3666 to (62.3, -34.89, -276.3) mm, rotated rx -152.51 ry -6.42 rz -112.51 deg; joints [10.856, -33.249, 94.254, 215.256, 109.876, 46.328, 26.033]
  MoveL 3667 to (62.26, -34.59, -276.2) mm, rotated rx -152.51 ry -6.42 rz -112.51 deg; joints [10.856, -33.247, 94.229, 215.251, 109.858, 46.314, 26.033]
  MoveL 3668 to (62.32, -34.62, -276.01) mm, rotated rx -152.51 ry -6.42 rz -112.51 deg; joints [10.855, -33.233, 94.214, 215.25, 109.857, 46.314, 26.033]
  MoveL 3669 to (62.45, -35.03, -275.7) mm, rotated rx -152.51 ry -6.42 rz -112.51 deg; joints [10.854, -33.206, 94.209, 215.254, 109.874, 46.327, 26.033]
  MoveL 3670 to (62.82, -35.12, -275.08) mm, rotated rx -152.51 ry -6.42 rz -112.51 deg; joints [10.845, -33.16, 94.16, 215.247, 109.869, 46.329, 26.033]
  MoveL 3671 to (62.89, -33.09, -275.07) mm, rotated rx -152.51 ry -6.42 rz -112.51 deg; joints [10.83, -33.182, 94.049, 215.208, 109.756, 46.254, 26.033]
  MoveL 3672 to (63.04, -30.95, -275.01) mm, rotated rx -152.51 ry -6.42 rz -112.51 deg; joints [10.812, -33.201, 93.927, 215.166, 109.637, 46.176, 26.033]
  MoveL 3673 to (63.25, -28.69, -274.89) mm, rotated rx -152.51 ry -6.42 rz -112.51 deg; joints [10.792, -33.216, 93.793, 215.121, 109.509, 46.093, 26.033]
  MoveL 3674 to (63.44, -26.46, -274.79) mm, rotated rx -152.51 ry -6.42 rz -112.51 deg; joints [10.772, -33.231, 93.662, 215.076, 109.383, 46.012, 26.033]
  MoveL 3675 to (63.64, -24.32, -274.62) mm, rotated rx -152.51 ry -6.42 rz -112.51 deg; joints [10.752, -33.24, 93.528, 215.034, 109.261, 45.934, 26.033]
  MoveL 3676 to (63.82, -22.38, -274.47) mm, rotated rx -152.51 ry -6.42 rz -112.51 deg; joints [10.735, -33.249, 93.409, 214.995, 109.151, 45.863, 26.033]
  MoveL 3677 to (64, -20.32, -274.42) mm, rotated rx -152.51 ry -6.42 rz -112.51 deg; joints [10.716, -33.265, 93.29, 214.955, 109.035, 45.789, 26.033]
  MoveL 3678 to (64.19, -18.17, -274.35) mm, rotated rx -152.51 ry -6.42 rz -112.51 deg; joints [10.697, -33.281, 93.164, 214.913, 108.914, 45.712, 26.033]
  MoveL 3679 to (64.4, -15.83, -274.19) mm, rotated rx -152.51 ry -6.42 rz -112.51 deg; joints [10.677, -33.292, 93.02, 214.868, 108.78, 45.627, 26.033]
  MoveL 3680 to (64.56, -13.96, -274.08) mm, rotated rx -152.51 ry -6.42 rz -112.51 deg; joints [10.66, -33.301, 92.905, 214.832, 108.673, 45.559, 26.033]
  MoveL 3681 to (64.76, -11.58, -273.87) mm, rotated rx -152.51 ry -6.42 rz -112.51 deg; joints [10.64, -33.308, 92.753, 214.787, 108.537, 45.472, 26.033]
  MoveL 3682 to (64.92, -9.71, -273.75) mm, rotated rx -152.51 ry -6.42 rz -112.51 deg; joints [10.624, -33.317, 92.637, 214.752, 108.43, 45.405, 26.033]
  MoveL 3683 to (65.09, -7.58, -273.59) mm, rotated rx -152.51 ry -6.42 rz -112.51 deg; joints [10.606, -33.325, 92.502, 214.712, 108.308, 45.327, 26.033]
  MoveL 3684 to (65.29, -5.2, -273.54) mm, rotated rx -152.51 ry -6.42 rz -112.51 deg; joints [10.585, -33.341, 92.363, 214.668, 108.174, 45.243, 26.033]
  MoveL 3685 to (65.44, -3.33, -273.42) mm, rotated rx -152.51 ry -6.42 rz -112.51 deg; joints [10.57, -33.349, 92.246, 214.633, 108.067, 45.176, 26.033]
  MoveL 3686 to (65.6, -1.2, -273.26) mm, rotated rx -152.51 ry -6.42 rz -112.51 deg; joints [10.552, -33.356, 92.111, 214.594, 107.944, 45.099, 26.033]
  MoveL 3687 to (65.79, 1.18, -273.21) mm, rotated rx -152.51 ry -6.42 rz -112.51 deg; joints [10.531, -33.371, 91.97, 214.551, 107.81, 45.015, 26.033]
  MoveL 3688 to (65.94, 3.05, -273.1) mm, rotated rx -152.51 ry -6.42 rz -112.51 deg; joints [10.516, -33.378, 91.852, 214.517, 107.702, 44.947, 26.033]
  MoveL 3689 to (66.11, 5.27, -273) mm, rotated rx -152.51 ry -6.42 rz -112.51 deg; joints [10.497, -33.389, 91.715, 214.478, 107.575, 44.868, 26.033]
  MoveL 3690 to (66.28, 7.49, -272.93) mm, rotated rx -152.51 ry -6.42 rz -112.51 deg; joints [10.479, -33.401, 91.581, 214.438, 107.449, 44.79, 26.033]
  MoveL 3691 to (66.4, 9.37, -272.75) mm, rotated rx -152.51 ry -6.42 rz -112.51 deg; joints [10.465, -33.403, 91.456, 214.406, 107.34, 44.721, 26.033]
  MoveL 3692 to (66.48, 11.1, -272.5) mm, rotated rx -152.51 ry -6.42 rz -112.51 deg; joints [10.453, -33.399, 91.333, 214.376, 107.239, 44.656, 26.033]
  MoveL 3693 to (66.52, 12.72, -272.14) mm, rotated rx -152.51 ry -6.42 rz -112.51 deg; joints [10.444, -33.388, 91.208, 214.35, 107.142, 44.593, 26.033]
  MoveL 3694 to (65.98, 11.32, -271.45) mm, rotated rx -152.51 ry -6.42 rz -112.51 deg; joints [10.474, -33.336, 91.232, 214.384, 107.213, 44.623, 26.033]
  MoveL 3695 to (66.04, 11.54, -271.45) mm, rotated rx -152.51 ry -6.42 rz -112.51 deg; joints [10.471, -33.337, 91.218, 214.38, 107.2, 44.616, 26.033]
  MoveL 3696 to (66.16, 11.81, -271.44) mm, rotated rx -152.51 ry -6.42 rz -112.51 deg; joints [10.465, -33.337, 91.201, 214.373, 107.184, 44.608, 26.033]
  MoveL 3697 to (66.4, 12.2, -271.41) mm, rotated rx -152.51 ry -6.42 rz -112.51 deg; joints [10.455, -33.336, 91.175, 214.361, 107.16, 44.599, 26.033]
  MoveL 3698 to (66.7, 12.64, -271.37) mm, rotated rx -152.51 ry -6.42 rz -112.51 deg; joints [10.442, -33.333, 91.145, 214.347, 107.134, 44.588, 26.033]
  MoveL 3699 to (67.06, 13.14, -271.32) mm, rotated rx -152.51 ry -6.42 rz -112.51 deg; joints [10.427, -33.33, 91.111, 214.331, 107.104, 44.577, 26.033]
  MoveL 3700 to (68.69, 15.19, -271.32) mm, rotated rx -152.51 ry -6.42 rz -112.51 deg; joints [10.358, -33.328, 90.986, 214.261, 106.982, 44.537, 26.033]
  MoveL 3701 to (69.06, 15.67, -271.29) mm, rotated rx -152.51 ry -6.42 rz -112.51 deg; joints [10.343, -33.325, 90.954, 214.245, 106.953, 44.526, 26.033]
  MoveL 3702 to (69.46, 16.23, -271.23) mm, rotated rx -152.51 ry -6.42 rz -112.51 deg; joints [10.326, -33.321, 90.915, 214.227, 106.92, 44.514, 26.033]
  MoveL 3703 to (69.84, 16.73, -271.2) mm, rotated rx -152.51 ry -6.42 rz -112.51 deg; joints [10.311, -33.318, 90.882, 214.211, 106.889, 44.503, 26.033]
  MoveL 3704 to (70.17, 17.14, -271.2) mm, rotated rx -152.51 ry -6.42 rz -112.51 deg; joints [10.297, -33.318, 90.857, 214.197, 106.865, 44.495, 26.033]
  MoveL 3705 to (70.47, 17.52, -271.2) mm, rotated rx -152.51 ry -6.42 rz -112.51 deg; joints [10.284, -33.317, 90.833, 214.184, 106.842, 44.487, 26.033]
  MoveL 3706 to (70.8, 17.93, -271.2) mm, rotated rx -152.51 ry -6.42 rz -112.51 deg; joints [10.271, -33.316, 90.807, 214.17, 106.818, 44.479, 26.033]
  MoveL 3707 to (71.12, 18.34, -271.19) mm, rotated rx -152.51 ry -6.42 rz -112.51 deg; joints [10.257, -33.315, 90.782, 214.157, 106.794, 44.471, 26.033]
  MoveL 3708 to (71.42, 18.72, -271.17) mm, rotated rx -152.51 ry -6.42 rz -112.51 deg; joints [10.245, -33.313, 90.757, 214.144, 106.77, 44.463, 26.033]
  MoveL 3709 to (71.69, 19.1, -271.12) mm, rotated rx -152.51 ry -6.42 rz -112.51 deg; joints [10.234, -33.309, 90.73, 214.132, 106.747, 44.455, 26.033]
  MoveL 3710 to (71.99, 19.49, -271.1) mm, rotated rx -152.51 ry -6.42 rz -112.51 deg; joints [10.221, -33.308, 90.704, 214.119, 106.724, 44.446, 26.033]
  MoveL 3711 to (72.32, 19.9, -271.1) mm, rotated rx -152.51 ry -6.42 rz -112.51 deg; joints [10.207, -33.307, 90.678, 214.105, 106.699, 44.438, 26.033]
  MoveL 3712 to (72.98, 20.72, -271.1) mm, rotated rx -152.51 ry -6.42 rz -112.51 deg; joints [10.18, -33.305, 90.628, 214.078, 106.65, 44.422, 26.033]
  Set speed (1000.0 mm/s)
  MoveL 3713 to (90.69, 33.12, -271.1) mm, rotated rx -152.51 ry -6.42 rz -112.51 deg; joints [9.503, -33.186, 89.82, 213.488, 105.874, 44.343, 26.033]
  Print: /'Flow1'
  Set speed (1000.0 mm/s)
  MoveL 3714 to (-65.26, 87.93, -71.64) mm, rotated rx -167.81 ry 3.47 rz -52.11 deg; joints [3.069, -25.408, 91.165, 149.611, 93.547, 27.414, -1.714]
  Set speed (1000.0 mm/s)
  MoveL 3715 to (-61.35, 43.22, -71.64) mm, rotated rx -167.81 ry 3.47 rz -52.11 deg; joints [3.131, -25.982, 94.841, 149.533, 96.21, 25.816, -1.714]
  Set speed (100.0 mm/s)
  MoveL 3716 to (-55, -29.26, -71.64) mm, rotated rx -167.81 ry 3.47 rz -52.11 deg; joints [3.24, -26.563, 100.416, 149.258, 100.491, 23.217, -1.714]
  MoveL 3717 to (-55.29, -29.7, -71.64) mm, rotated rx -167.81 ry 3.47 rz -52.11 deg; joints [3.252, -26.571, 100.451, 149.267, 100.513, 23.2, -1.714]
  MoveL 3718 to (-55.59, -30.27, -71.55) mm, rotated rx -167.81 ry 3.47 rz -52.11 deg; joints [3.267, -26.574, 100.49, 149.277, 100.541, 23.178, -1.714]
  MoveL 3719 to (-55.89, -30.78, -71.49) mm, rotated rx -167.81 ry 3.47 rz -52.11 deg; joints [3.281, -26.58, 100.528, 149.287, 100.567, 23.158, -1.714]
  MoveL 3720 to (-56.19, -31.26, -71.47) mm, rotated rx -167.81 ry 3.47 rz -52.11 deg; joints [3.295, -26.587, 100.565, 149.297, 100.59, 23.139, -1.714]
  MoveL 3721 to (-58.19, -34.33, -71.47) mm, rotated rx -167.81 ry 3.47 rz -52.11 deg; joints [3.384, -26.644, 100.809, 149.36, 100.739, 23.02, -1.714]
  MoveL 3722 to (-59.04, -35.52, -71.56) mm, rotated rx -167.81 ry 3.47 rz -52.11 deg; joints [3.42, -26.673, 100.909, 149.386, 100.795, 22.975, -1.714]
  MoveL 3723 to (-59.83, -36.4, -71.82) mm, rotated rx -167.81 ry 3.47 rz -52.11 deg; joints [3.451, -26.71, 100.997, 149.41, 100.835, 22.941, -1.714]
  MoveL 3724 to (-60.57, -36.98, -72.27) mm, rotated rx -167.81 ry 3.47 rz -52.11 deg; joints [3.476, -26.756, 101.073, 149.43, 100.857, 22.92, -1.714]
  MoveL 3725 to (-60.93, -37.17, -72.56) mm, rotated rx -167.81 ry 3.47 rz -52.11 deg; joints [3.487, -26.782, 101.106, 149.439, 100.862, 22.913, -1.714]
  MoveL 3726 to (-61.27, -37.27, -72.89) mm, rotated rx -167.81 ry 3.47 rz -52.11 deg; joints [3.496, -26.811, 101.137, 149.448, 100.862, 22.91, -1.714]
  MoveL 3727 to (-61.91, -37.26, -73.69) mm, rotated rx -167.81 ry 3.47 rz -52.11 deg; joints [3.511, -26.874, 101.189, 149.463, 100.85, 22.912, -1.714]
  MoveL 3728 to (-62.51, -36.96, -74.66) mm, rotated rx -167.81 ry 3.47 rz -52.11 deg; joints [3.521, -26.946, 101.229, 149.475, 100.821, 22.927, -1.714]
  MoveL 3729 to (-63.55, -35.46, -77.15) mm, rotated rx -167.81 ry 3.47 rz -52.11 deg; joints [3.525, -27.116, 101.274, 149.49, 100.713, 22.991, -1.714]
  MoveL 3730 to (-64.12, -33.31, -79.63) mm, rotated rx -167.81 ry 3.47 rz -52.11 deg; joints [3.508, -27.273, 101.266, 149.49, 100.574, 23.08, -1.714]
  MoveL 3731 to (-63.95, -31.09, -81.41) mm, rotated rx -167.81 ry 3.47 rz -52.11 deg; joints [3.471, -27.37, 101.204, 149.471, 100.442, 23.171, -1.714]
  MoveL 3732 to (-63.59, -29.94, -82.03) mm, rotated rx -167.81 ry 3.47 rz -52.11 deg; joints [3.445, -27.396, 101.153, 149.455, 100.379, 23.217, -1.714]
  MoveL 3733 to (-63.04, -28.77, -82.47) mm, rotated rx -167.81 ry 3.47 rz -52.11 deg; joints [3.414, -27.406, 101.088, 149.433, 100.318, 23.264, -1.714]
  MoveL 3734 to (-61.38, -26.37, -82.83) mm, rotated rx -167.81 ry 3.47 rz -52.11 deg; joints [3.337, -27.382, 100.916, 149.377, 100.203, 23.359, -1.714]
  MoveL 3735 to (-59.37, -23.95, -82.83) mm, rotated rx -167.81 ry 3.47 rz -52.11 deg; joints [3.251, -27.328, 100.719, 149.311, 100.092, 23.454, -1.714]
  MoveL 3736 to (-59.07, -23.56, -82.85) mm, rotated rx -167.81 ry 3.47 rz -52.11 deg; joints [3.238, -27.321, 100.689, 149.301, 100.074, 23.469, -1.714]
  MoveL 3737 to (-58.8, -23.2, -82.89) mm, rotated rx -167.81 ry 3.47 rz -52.11 deg; joints [3.226, -27.316, 100.661, 149.292, 100.057, 23.484, -1.714]
  MoveL 3738 to (-58.56, -22.85, -82.95) mm, rotated rx -167.81 ry 3.47 rz -52.11 deg; joints [3.215, -27.313, 100.637, 149.284, 100.04, 23.498, -1.714]
  MoveL 3739 to (-58.3, -22.49, -83) mm, rotated rx -167.81 ry 3.47 rz -52.11 deg; joints [3.203, -27.309, 100.611, 149.275, 100.023, 23.512, -1.714]
  MoveL 3740 to (-57.97, -22.06, -83.03) mm, rotated rx -167.81 ry 3.47 rz -52.11 deg; joints [3.188, -27.301, 100.577, 149.264, 100.003, 23.529, -1.714]
  MoveL 3741 to (-57.57, -21.55, -83.07) mm, rotated rx -167.81 ry 3.47 rz -52.11 deg; joints [3.171, -27.292, 100.538, 149.251, 99.979, 23.55, -1.714]
  MoveL 3742 to (-57.24, -21.09, -83.13) mm, rotated rx -167.81 ry 3.47 rz -52.11 deg; joints [3.156, -27.286, 100.505, 149.24, 99.958, 23.568, -1.714]
  MoveL 3743 to (-56.98, -20.72, -83.2) mm, rotated rx -167.81 ry 3.47 rz -52.11 deg; joints [3.144, -27.284, 100.479, 149.231, 99.94, 23.583, -1.714]
  MoveL 3744 to (-56.73, -20.37, -83.25) mm, rotated rx -167.81 ry 3.47 rz -52.11 deg; joints [3.132, -27.28, 100.453, 149.222, 99.923, 23.597, -1.714]
  MoveL 3745 to (-56.44, -19.99, -83.27) mm, rotated rx -167.81 ry 3.47 rz -52.11 deg; joints [3.12, -27.273, 100.424, 149.213, 99.905, 23.612, -1.714]
  MoveL 3746 to (-56.1, -19.59, -83.27) mm, rotated rx -167.81 ry 3.47 rz -52.11 deg; joints [3.105, -27.264, 100.391, 149.202, 99.887, 23.628, -1.714]
  MoveL 3747 to (-55.76, -19.17, -83.27) mm, rotated rx -167.81 ry 3.47 rz -52.11 deg; joints [3.091, -27.254, 100.357, 149.191, 99.868, 23.644, -1.714]
  MoveL 3748 to (-55.4, -18.73, -83.29) mm, rotated rx -167.81 ry 3.47 rz -52.11 deg; joints [3.076, -27.245, 100.321, 149.179, 99.847, 23.662, -1.714]
  MoveL 3749 to (-55.01, -18.2, -83.32) mm, rotated rx -167.81 ry 3.47 rz -52.11 deg; joints [3.058, -27.236, 100.279, 149.166, 99.822, 23.683, -1.714]
  MoveL 3750 to (-54.68, -17.7, -83.38) mm, rotated rx -167.81 ry 3.47 rz -52.11 deg; joints [3.043, -27.23, 100.243, 149.155, 99.798, 23.703, -1.714]
  MoveL 3751 to (-54.45, -17.31, -83.49) mm, rotated rx -167.81 ry 3.47 rz -52.11 deg; joints [3.032, -27.229, 100.218, 149.147, 99.779, 23.719, -1.714]
  MoveL 3752 to (-54.44, -17.31, -83.72) mm, rotated rx -167.81 ry 3.47 rz -52.11 deg; joints [3.029, -27.245, 100.232, 149.144, 99.778, 23.72, -1.714]
  MoveL 3753 to (-54.58, -17.69, -84.08) mm, rotated rx -167.81 ry 3.47 rz -52.11 deg; joints [3.032, -27.273, 100.282, 149.145, 99.796, 23.708, -1.714]
  MoveL 3754 to (-55.4, -17.92, -85.04) mm, rotated rx -167.81 ry 3.47 rz -52.11 deg; joints [3.052, -27.352, 100.363, 149.163, 99.795, 23.701, -1.714]
  MoveL 3755 to (-55.18, -15.8, -85.04) mm, rotated rx -167.81 ry 3.47 rz -52.11 deg; joints [3.034, -27.331, 100.201, 149.16, 99.676, 23.78, -1.714]
  MoveL 3756 to (-54.98, -13.51, -85.17) mm, rotated rx -167.81 ry 3.47 rz -52.11 deg; joints [3.015, -27.318, 100.034, 149.155, 99.547, 23.865, -1.714]
  MoveL 3757 to (-54.77, -11.34, -85.23) mm, rotated rx -167.81 ry 3.47 rz -52.11 deg; joints [2.997, -27.3, 99.871, 149.151, 99.426, 23.945, -1.714]
  MoveL 3758 to (-54.57, -9.23, -85.36) mm, rotated rx -167.81 ry 3.47 rz -52.11 deg; joints [2.978, -27.287, 99.716, 149.146, 99.306, 24.023, -1.714]
  MoveL 3759 to (-54.38, -7.1, -85.52) mm, rotated rx -167.81 ry 3.47 rz -52.11 deg; joints [2.96, -27.276, 99.561, 149.141, 99.186, 24.103, -1.714]
  MoveL 3760 to (-54.17, -4.98, -85.64) mm, rotated rx -167.81 ry 3.47 rz -52.11 deg; joints [2.941, -27.262, 99.405, 149.136, 99.067, 24.182, -1.714]
  MoveL 3761 to (-53.97, -2.85, -85.85) mm, rotated rx -167.81 ry 3.47 rz -52.11 deg; joints [2.922, -27.253, 99.252, 149.131, 98.946, 24.262, -1.714]
  MoveL 3762 to (-53.77, -0.73, -85.96) mm, rotated rx -167.81 ry 3.47 rz -52.11 deg; joints [2.904, -27.237, 99.095, 149.125, 98.828, 24.34, -1.714]
  MoveL 3763 to (-53.55, 1.4, -86.02) mm, rotated rx -167.81 ry 3.47 rz -52.11 deg; joints [2.886, -27.218, 98.932, 149.12, 98.708, 24.419, -1.714]
  MoveL 3764 to (-53.33, 3.55, -86.17) mm, rotated rx -167.81 ry 3.47 rz -52.11 deg; joints [2.867, -27.203, 98.773, 149.114, 98.587, 24.499, -1.714]
  MoveL 3765 to (-53.11, 5.76, -86.35) mm, rotated rx -167.81 ry 3.47 rz -52.11 deg; joints [2.847, -27.19, 98.61, 149.107, 98.462, 24.582, -1.714]
  MoveL 3766 to (-52.88, 7.98, -86.53) mm, rotated rx -167.81 ry 3.47 rz -52.11 deg; joints [2.826, -27.175, 98.447, 149.1, 98.338, 24.665, -1.714]
  MoveL 3767 to (-52.68, 9.84, -86.77) mm, rotated rx -167.81 ry 3.47 rz -52.11 deg; joints [2.808, -27.169, 98.315, 149.093, 98.233, 24.736, -1.714]
  MoveL 3768 to (-52.4, 12.49, -86.87) mm, rotated rx -167.81 ry 3.47 rz -52.11 deg; joints [2.785, -27.144, 98.112, 149.086, 98.084, 24.835, -1.714]
  Set speed (1000.0 mm/s)
  MoveL 3769 to (-56.35, 57.63, -86.87) mm, rotated rx -167.81 ry 3.47 rz -52.11 deg; joints [2.731, -26.679, 94.537, 149.225, 95.423, 26.457, -1.714]
  Set speed (1000.0 mm/s)
  MoveL 3770 to (-50.64, 58.13, -98.75) mm, rotated rx -167.81 ry 3.47 rz -52.11 deg; joints [2.401, -27.328, 95.144, 148.932, 95.451, 26.586, -1.714]
  Set speed (100.0 mm/s)
  MoveL 3771 to (-48.14, 29.55, -98.75) mm, rotated rx -167.81 ry 3.47 rz -52.11 deg; joints [2.429, -27.644, 97.427, 148.846, 97.131, 25.554, -1.714]
  MoveL 3772 to (-48.55, 27.88, -98.51) mm, rotated rx -167.81 ry 3.47 rz -52.11 deg; joints [2.454, -27.655, 97.549, 148.86, 97.221, 25.489, -1.714]
  MoveL 3773 to (-49, 25.91, -98.44) mm, rotated rx -167.81 ry 3.47 rz -52.11 deg; joints [2.479, -27.681, 97.705, 148.874, 97.328, 25.414, -1.714]
  MoveL 3774 to (-49.46, 23.9, -98.3) mm, rotated rx -167.81 ry 3.47 rz -52.11 deg; joints [2.505, -27.702, 97.859, 148.889, 97.436, 25.337, -1.714]
  MoveL 3775 to (-50.02, 21.51, -98.16) mm, rotated rx -167.81 ry 3.47 rz -52.11 deg; joints [2.537, -27.73, 98.044, 148.907, 97.566, 25.246, -1.714]
  MoveL 3776 to (-50.49, 19.43, -98.16) mm, rotated rx -167.81 ry 3.47 rz -52.11 deg; joints [2.563, -27.761, 98.212, 148.921, 97.678, 25.167, -1.714]
  MoveL 3777 to (-51.01, 17.12, -98.01) mm, rotated rx -167.81 ry 3.47 rz -52.11 deg; joints [2.593, -27.785, 98.388, 148.938, 97.803, 25.079, -1.714]
  MoveL 3778 to (-51.45, 15.18, -97.82) mm, rotated rx -167.81 ry 3.47 rz -52.11 deg; joints [2.619, -27.801, 98.533, 148.953, 97.909, 25.005, -1.714]
  MoveL 3779 to (-51.91, 13.19, -97.73) mm, rotated rx -167.81 ry 3.47 rz -52.11 deg; joints [2.646, -27.824, 98.687, 148.967, 98.017, 24.929, -1.714]
  MoveL 3780 to (-52.38, 11.11, -97.51) mm, rotated rx -167.81 ry 3.47 rz -52.11 deg; joints [2.674, -27.84, 98.841, 148.982, 98.13, 24.849, -1.714]
  MoveL 3781 to (-52.83, 9.04, -97.35) mm, rotated rx -167.81 ry 3.47 rz -52.11 deg; joints [2.701, -27.859, 98.995, 148.997, 98.243, 24.771, -1.714]
  MoveL 3782 to (-53.29, 6.98, -97.24) mm, rotated rx -167.81 ry 3.47 rz -52.11 deg; joints [2.728, -27.88, 99.153, 149.011, 98.355, 24.692, -1.714]
  MoveL 3783 to (-53.74, 4.89, -97.08) mm, rotated rx -167.81 ry 3.47 rz -52.11 deg; joints [2.755, -27.898, 99.309, 149.025, 98.469, 24.613, -1.714]
  MoveL 3784 to (-54.2, 2.81, -96.93) mm, rotated rx -167.81 ry 3.47 rz -52.11 deg; joints [2.783, -27.917, 99.465, 149.04, 98.582, 24.534, -1.714]
  MoveL 3785 to (-54.67, 0.68, -96.87) mm, rotated rx -167.81 ry 3.47 rz -52.11 deg; joints [2.81, -27.941, 99.629, 149.053, 98.697, 24.454, -1.714]
  MoveL 3786 to (-55.11, -1.4, -96.66) mm, rotated rx -167.81 ry 3.47 rz -52.11 deg; joints [2.837, -27.955, 99.781, 149.068, 98.811, 24.374, -1.714]
  MoveL 3787 to (-55.55, -3.48, -96.53) mm, rotated rx -167.81 ry 3.47 rz -52.11 deg; joints [2.864, -27.974, 99.936, 149.081, 98.924, 24.296, -1.714]
  MoveL 3788 to (-56, -5.59, -96.41) mm, rotated rx -167.81 ry 3.47 rz -52.11 deg; joints [2.892, -27.993, 100.095, 149.095, 99.039, 24.216, -1.714]
  MoveL 3789 to (-56.24, -7.35, -96.2) mm, rotated rx -167.81 ry 3.47 rz -52.11 deg; joints [2.911, -27.999, 100.219, 149.102, 99.137, 24.15, -1.714]
  MoveL 3790 to (-56.31, -8.82, -95.85) mm, rotated rx -167.81 ry 3.47 rz -52.11 deg; joints [2.924, -27.99, 100.311, 149.106, 99.222, 24.094, -1.714]
  MoveL 3791 to (-56.17, -10.02, -95.33) mm, rotated rx -167.81 ry 3.47 rz -52.11 deg; joints [2.93, -27.964, 100.371, 149.104, 99.295, 24.048, -1.714]
  MoveL 3792 to (-55.4, -8.69, -94.47) mm, rotated rx -167.81 ry 3.47 rz -52.11 deg; joints [2.905, -27.884, 100.214, 149.088, 99.233, 24.094, -1.714]
  MoveL 3793 to (-55.74, -9.42, -94.47) mm, rotated rx -167.81 ry 3.47 rz -52.11 deg; joints [2.921, -27.896, 100.272, 149.098, 99.27, 24.066, -1.714]
  MoveL 3794 to (-56.09, -10.03, -94.47) mm, rotated rx -167.81 ry 3.47 rz -52.11 deg; joints [2.937, -27.908, 100.321, 149.11, 99.3, 24.042, -1.714]
  MoveL 3795 to (-56.49, -10.52, -94.46) mm, rotated rx -167.81 ry 3.47 rz -52.11 deg; joints [2.954, -27.919, 100.362, 149.123, 99.322, 24.023, -1.714]
  MoveL 3796 to (-56.94, -11.01, -94.44) mm, rotated rx -167.81 ry 3.47 rz -52.11 deg; joints [2.973, -27.93, 100.402, 149.137, 99.344, 24.003, -1.714]
  MoveL 3797 to (-57.47, -11.56, -94.41) mm, rotated rx -167.81 ry 3.47 rz -52.11 deg; joints [2.995, -27.942, 100.446, 149.155, 99.368, 23.98, -1.714]
  MoveL 3798 to (-58.99, -13, -94.41) mm, rotated rx -167.81 ry 3.47 rz -52.11 deg; joints [3.057, -27.982, 100.567, 149.205, 99.429, 23.921, -1.714]
  MoveL 3799 to (-59.31, -13.32, -94.39) mm, rotated rx -167.81 ry 3.47 rz -52.11 deg; joints [3.071, -27.989, 100.592, 149.216, 99.442, 23.909, -1.714]
  MoveL 3800 to (-60.07, -14.04, -94.39) mm, rotated rx -167.81 ry 3.47 rz -52.11 deg; joints [3.102, -28.009, 100.653, 149.241, 99.472, 23.879, -1.714]
  MoveL 3801 to (-60.43, -14.39, -94.39) mm, rotated rx -167.81 ry 3.47 rz -52.11 deg; joints [3.117, -28.018, 100.682, 149.253, 99.487, 23.865, -1.714]
  MoveL 3802 to (-60.78, -14.73, -94.37) mm, rotated rx -167.81 ry 3.47 rz -52.11 deg; joints [3.132, -28.026, 100.71, 149.264, 99.502, 23.851, -1.714]
  MoveL 3803 to (-61.11, -15.08, -94.33) mm, rotated rx -167.81 ry 3.47 rz -52.11 deg; joints [3.146, -28.033, 100.737, 149.276, 99.517, 23.837, -1.714]
  MoveL 3804 to (-61.4, -15.4, -94.28) mm, rotated rx -167.81 ry 3.47 rz -52.11 deg; joints [3.159, -28.037, 100.76, 149.286, 99.532, 23.824, -1.714]
  MoveL 3805 to (-61.73, -15.75, -94.24) mm, rotated rx -167.81 ry 3.47 rz -52.11 deg; joints [3.173, -28.043, 100.787, 149.297, 99.547, 23.81, -1.714]
  MoveL 3806 to (-62.08, -16.09, -94.22) mm, rotated rx -167.81 ry 3.47 rz -52.11 deg; joints [3.187, -28.051, 100.815, 149.308, 99.562, 23.796, -1.714]
  MoveL 3807 to (-62.44, -16.45, -94.21) mm, rotated rx -167.81 ry 3.47 rz -52.11 deg; joints [3.203, -28.06, 100.844, 149.32, 99.577, 23.781, -1.714]
  MoveL 3808 to (-62.79, -16.8, -94.19) mm, rotated rx -167.81 ry 3.47 rz -52.11 deg; joints [3.217, -28.068, 100.872, 149.332, 99.592, 23.767, -1.714]
  MoveL 3809 to (-63.12, -17.15, -94.16) mm, rotated rx -167.81 ry 3.47 rz -52.11 deg; joints [3.231, -28.075, 100.899, 149.343, 99.607, 23.753, -1.714]
  MoveL 3810 to (-63.4, -17.48, -94.1) mm, rotated rx -167.81 ry 3.47 rz -52.11 deg; joints [3.244, -28.079, 100.922, 149.353, 99.622, 23.74, -1.714]
  MoveL 3811 to (-63.7, -17.82, -94.05) mm, rotated rx -167.81 ry 3.47 rz -52.11 deg; joints [3.257, -28.084, 100.947, 149.363, 99.638, 23.726, -1.714]
  MoveL 3812 to (-64.7, -18.86, -93.96) mm, rotated rx -167.81 ry 3.47 rz -52.11 deg; joints [3.3, -28.105, 101.028, 149.397, 99.683, 23.684, -1.714]
  MoveL 3813 to (-65.61, -19.6, -94.09) mm, rotated rx -167.81 ry 3.47 rz -52.11 deg; joints [3.336, -28.135, 101.099, 149.426, 99.712, 23.654, -1.714]
  MoveL 3814 to (-66.45, -20.04, -94.43) mm, rotated rx -167.81 ry 3.47 rz -52.11 deg; joints [3.365, -28.176, 101.158, 149.451, 99.723, 23.637, -1.714]
  MoveL 3815 to (-66.83, -20.15, -94.68) mm, rotated rx -167.81 ry 3.47 rz -52.11 deg; joints [3.377, -28.2, 101.183, 149.462, 99.723, 23.633, -1.714]
  MoveL 3816 to (-67.2, -20.19, -94.98) mm, rotated rx -167.81 ry 3.47 rz -52.11 deg; joints [3.387, -28.226, 101.206, 149.472, 99.719, 23.632, -1.714]
  MoveL 3817 to (-67.87, -20.04, -95.73) mm, rotated rx -167.81 ry 3.47 rz -52.11 deg; joints [3.403, -28.286, 101.244, 149.488, 99.697, 23.64, -1.714]
  MoveL 3818 to (-68.45, -19.59, -96.7) mm, rotated rx -167.81 ry 3.47 rz -52.11 deg; joints [3.411, -28.355, 101.27, 149.5, 99.659, 23.66, -1.714]
  MoveL 3819 to (-69.38, -17.8, -99.27) mm, rotated rx -167.81 ry 3.47 rz -52.11 deg; joints [3.408, -28.524, 101.29, 149.51, 99.531, 23.737, -1.714]
  MoveL 3820 to (-69.73, -15.49, -101.88) mm, rotated rx -167.81 ry 3.47 rz -52.11 deg; joints [3.381, -28.68, 101.268, 149.5, 99.382, 23.836, -1.714]
  MoveL 3821 to (-69.59, -14.37, -102.91) mm, rotated rx -167.81 ry 3.47 rz -52.11 deg; joints [3.359, -28.734, 101.241, 149.487, 99.315, 23.883, -1.714]
  MoveL 3822 to (-69.25, -13.29, -103.74) mm, rotated rx -167.81 ry 3.47 rz -52.11 deg; joints [3.332, -28.773, 101.205, 149.468, 99.255, 23.929, -1.714]
  MoveL 3823 to (-68.7, -12.24, -104.4) mm, rotated rx -167.81 ry 3.47 rz -52.11 deg; joints [3.3, -28.796, 101.158, 149.445, 99.2, 23.973, -1.714]
  MoveL 3824 to (-67.94, -11.22, -104.86) mm, rotated rx -167.81 ry 3.47 rz -52.11 deg; joints [3.262, -28.804, 101.102, 149.415, 99.15, 24.016, -1.714]
  MoveL 3825 to (-66.97, -10.23, -105.14) mm, rotated rx -167.81 ry 3.47 rz -52.11 deg; joints [3.219, -28.795, 101.036, 149.381, 99.107, 24.058, -1.714]
  MoveL 3826 to (-65.8, -9.27, -105.24) mm, rotated rx -167.81 ry 3.47 rz -52.11 deg; joints [3.17, -28.772, 100.959, 149.341, 99.069, 24.098, -1.714]
  MoveL 3827 to (-63.26, -7.39, -105.24) mm, rotated rx -167.81 ry 3.47 rz -52.11 deg; joints [3.068, -28.709, 100.797, 149.256, 98.999, 24.177, -1.714]
  MoveL 3828 to (-62.82, -7.05, -105.25) mm, rotated rx -167.81 ry 3.47 rz -52.11 deg; joints [3.05, -28.699, 100.769, 149.241, 98.987, 24.191, -1.714]
  MoveL 3829 to (-62.34, -6.67, -105.29) mm, rotated rx -167.81 ry 3.47 rz -52.11 deg; joints [3.03, -28.689, 100.737, 149.225, 98.971, 24.207, -1.714]
  MoveL 3830 to (-61.76, -6.17, -105.38) mm, rotated rx -167.81 ry 3.47 rz -52.11 deg; joints [3.006, -28.68, 100.7, 149.205, 98.951, 24.228, -1.714]
  MoveL 3831 to (-61.28, -5.78, -105.42) mm, rotated rx -167.81 ry 3.47 rz -52.11 deg; joints [2.986, -28.67, 100.669, 149.189, 98.936, 24.245, -1.714]
  MoveL 3832 to (-60.85, -5.45, -105.44) mm, rotated rx -167.81 ry 3.47 rz -52.11 deg; joints [2.968, -28.66, 100.641, 149.174, 98.923, 24.259, -1.714]
  MoveL 3833 to (-60.45, -5.14, -105.44) mm, rotated rx -167.81 ry 3.47 rz -52.11 deg; joints [2.952, -28.651, 100.615, 149.161, 98.912, 24.272, -1.714]
  MoveL 3834 to (-60.09, -4.86, -105.46) mm, rotated rx -167.81 ry 3.47 rz -52.11 deg; joints [2.938, -28.643, 100.592, 149.149, 98.901, 24.284, -1.714]
  MoveL 3835 to (-58.43, -3.63, -105.47) mm, rotated rx -167.81 ry 3.47 rz -52.11 deg; joints [2.871, -28.602, 100.485, 149.094, 98.855, 24.336, -1.714]
  MoveL 3836 to (-58.04, -3.31, -105.5) mm, rotated rx -167.81 ry 3.47 rz -52.11 deg; joints [2.855, -28.594, 100.459, 149.08, 98.842, 24.349, -1.714]
  MoveL 3837 to (-57.68, -3, -105.56) mm, rotated rx -167.81 ry 3.47 rz -52.11 deg; joints [2.84, -28.588, 100.436, 149.068, 98.829, 24.362, -1.714]
  MoveL 3838 to (-57.34, -2.68, -105.63) mm, rotated rx -167.81 ry 3.47 rz -52.11 deg; joints [2.826, -28.584, 100.413, 149.056, 98.816, 24.376, -1.714]
  MoveL 3839 to (-57, -2.33, -105.69) mm, rotated rx -167.81 ry 3.47 rz -52.11 deg; joints [2.811, -28.578, 100.387, 149.045, 98.801, 24.391, -1.714]
  MoveL 3840 to (-56.63, -1.93, -105.72) mm, rotated rx -167.81 ry 3.47 rz -52.11 deg; joints [2.795, -28.57, 100.354, 149.032, 98.783, 24.407, -1.714]
  MoveL 3841 to (-56.25, -1.37, -105.73) mm, rotated rx -167.81 ry 3.47 rz -52.11 deg; joints [2.779, -28.558, 100.309, 149.02, 98.757, 24.429, -1.714]
  MoveL 3842 to (-55.88, -0.7, -105.73) mm, rotated rx -167.81 ry 3.47 rz -52.11 deg; joints [2.762, -28.545, 100.254, 149.008, 98.723, 24.456, -1.714]
  MoveL 3843 to (-57.51, -1.74, -107.28) mm, rotated rx -167.81 ry 3.47 rz -52.11 deg; joints [2.809, -28.684, 100.436, 149.048, 98.752, 24.421, -1.714]
  MoveL 3844 to (-56.74, 0.5, -107.42) mm, rotated rx -167.81 ry 3.47 rz -52.11 deg; joints [2.77, -28.658, 100.266, 149.023, 98.635, 24.506, -1.714]
  MoveL 3845 to (-56.01, 2.61, -107.53) mm, rotated rx -167.81 ry 3.47 rz -52.11 deg; joints [2.732, -28.632, 100.104, 149, 98.525, 24.587, -1.714]
  MoveL 3846 to (-55.31, 4.65, -107.69) mm, rotated rx -167.81 ry 3.47 rz -52.11 deg; joints [2.696, -28.61, 99.95, 148.977, 98.417, 24.666, -1.714]
  MoveL 3847 to (-54.61, 6.66, -107.8) mm, rotated rx -167.81 ry 3.47 rz -52.11 deg; joints [2.661, -28.584, 99.794, 148.955, 98.312, 24.744, -1.714]
  MoveL 3848 to (-53.91, 8.68, -107.9) mm, rotated rx -167.81 ry 3.47 rz -52.11 deg; joints [2.625, -28.558, 99.638, 148.932, 98.206, 24.822, -1.714]
  MoveL 3849 to (-53.22, 10.7, -108.13) mm, rotated rx -167.81 ry 3.47 rz -52.11 deg; joints [2.589, -28.54, 99.488, 148.909, 98.1, 24.9, -1.714]
  MoveL 3850 to (-52.52, 12.72, -108.35) mm, rotated rx -167.81 ry 3.47 rz -52.11 deg; joints [2.552, -28.521, 99.338, 148.886, 97.994, 24.979, -1.714]
  MoveL 3851 to (-51.81, 14.73, -108.46) mm, rotated rx -167.81 ry 3.47 rz -52.11 deg; joints [2.517, -28.494, 99.182, 148.863, 97.889, 25.057, -1.714]
  MoveL 3852 to (-51.09, 16.74, -108.46) mm, rotated rx -167.81 ry 3.47 rz -52.11 deg; joints [2.482, -28.46, 99.019, 148.841, 97.785, 25.134, -1.714]
  MoveL 3853 to (-50.38, 18.76, -108.58) mm, rotated rx -167.81 ry 3.47 rz -52.11 deg; joints [2.447, -28.433, 98.862, 148.818, 97.68, 25.212, -1.714]
  MoveL 3854 to (-49.66, 20.79, -108.78) mm, rotated rx -167.81 ry 3.47 rz -52.11 deg; joints [2.41, -28.41, 98.707, 148.794, 97.573, 25.292, -1.714]
  MoveL 3855 to (-48.98, 22.69, -108.96) mm, rotated rx -167.81 ry 3.47 rz -52.11 deg; joints [2.376, -28.389, 98.562, 148.771, 97.474, 25.366, -1.714]
  MoveL 3856 to (-48.35, 24.44, -109.18) mm, rotated rx -167.81 ry 3.47 rz -52.11 deg; joints [2.344, -28.372, 98.432, 148.75, 97.382, 25.435, -1.714]
  MoveL 3857 to (-47.69, 26.29, -109.27) mm, rotated rx -167.81 ry 3.47 rz -52.11 deg; joints [2.311, -28.345, 98.285, 148.729, 97.286, 25.507, -1.714]
  MoveL 3858 to (-46.99, 28.26, -109.28) mm, rotated rx -167.81 ry 3.47 rz -52.11 deg; joints [2.278, -28.31, 98.124, 148.707, 97.183, 25.583, -1.714]
  MoveL 3859 to (-46.06, 30.8, -109.38) mm, rotated rx -167.81 ry 3.47 rz -52.11 deg; joints [2.233, -28.27, 97.919, 148.677, 97.051, 25.683, -1.714]
  MoveL 3860 to (-45.36, 32.71, -109.59) mm, rotated rx -167.81 ry 3.47 rz -52.11 deg; joints [2.198, -28.248, 97.774, 148.654, 96.952, 25.758, -1.714]
  MoveL 3861 to (-44.58, 34.78, -109.79) mm, rotated rx -167.81 ry 3.47 rz -52.11 deg; joints [2.16, -28.222, 97.614, 148.628, 96.844, 25.84, -1.714]
  MoveL 3862 to (-43.86, 36.67, -110.08) mm, rotated rx -167.81 ry 3.47 rz -52.11 deg; joints [2.124, -28.205, 97.473, 148.603, 96.746, 25.916, -1.714]
  MoveL 3863 to (-43.18, 38.53, -110.2) mm, rotated rx -167.81 ry 3.47 rz -52.11 deg; joints [2.09, -28.178, 97.325, 148.58, 96.649, 25.989, -1.714]
  MoveL 3864 to (-42.47, 40.5, -110.22) mm, rotated rx -167.81 ry 3.47 rz -52.11 deg; joints [2.057, -28.142, 97.162, 148.558, 96.546, 26.066, -1.714]
  MoveL 3865 to (-41.83, 42.15, -110.45) mm, rotated rx -167.81 ry 3.47 rz -52.11 deg; joints [2.025, -28.124, 97.037, 148.536, 96.461, 26.132, -1.714]
  Set speed (1000.0 mm/s)
  MoveL 3866 to (-44.1, 68.11, -110.45) mm, rotated rx -167.81 ry 3.47 rz -52.11 deg; joints [2.006, -27.814, 94.94, 148.611, 94.94, 27.075, -1.714]
  Set speed (1000.0 mm/s)
  MoveL 3867 to (-37.59, 68.68, -121.64) mm, rotated rx -167.81 ry 3.47 rz -52.11 deg; joints [1.653, -28.398, 95.469, 148.299, 94.965, 27.221, -1.714]
  Set speed (100.0 mm/s)
  MoveL 3868 to (-35.83, 48.58, -121.64) mm, rotated rx -167.81 ry 3.47 rz -52.11 deg; joints [1.664, -28.644, 97.097, 148.239, 96.138, 26.487, -1.714]
  MoveL 3869 to (-36.79, 46.68, -121.64) mm, rotated rx -167.81 ry 3.47 rz -52.11 deg; joints [1.706, -28.686, 97.259, 148.269, 96.232, 26.411, -1.714]
  MoveL 3870 to (-37.82, 44.7, -121.54) mm, rotated rx -167.81 ry 3.47 rz -52.11 deg; joints [1.751, -28.724, 97.423, 148.302, 96.33, 26.33, -1.714]
  MoveL 3871 to (-38.94, 42.63, -121.25) mm, rotated rx -167.81 ry 3.47 rz -52.11 deg; joints [1.801, -28.753, 97.583, 148.34, 96.432, 26.245, -1.714]
  MoveL 3872 to (-40.01, 40.66, -120.9) mm, rotated rx -167.81 ry 3.47 rz -52.11 deg; joints [1.851, -28.775, 97.732, 148.377, 96.531, 26.163, -1.714]
  MoveL 3873 to (-40.97, 38.83, -120.71) mm, rotated rx -167.81 ry 3.47 rz -52.11 deg; joints [1.894, -28.803, 97.876, 148.409, 96.622, 26.088, -1.714]
  MoveL 3874 to (-41.87, 37.09, -120.57) mm, rotated rx -167.81 ry 3.47 rz -52.11 deg; joints [1.935, -28.832, 98.015, 148.438, 96.708, 26.018, -1.714]
  MoveL 3875 to (-42.8, 35.26, -120.52) mm, rotated rx -167.81 ry 3.47 rz -52.11 deg; joints [1.976, -28.869, 98.167, 148.468, 96.798, 25.945, -1.714]
  MoveL 3876 to (-43.76, 33.36, -120.5) mm, rotated rx -167.81 ry 3.47 rz -52.11 deg; joints [2.018, -28.908, 98.326, 148.498, 96.893, 25.869, -1.714]
  MoveL 3877 to (-44.73, 31.47, -120.39) mm, rotated rx -167.81 ry 3.47 rz -52.11 deg; joints [2.061, -28.94, 98.478, 148.53, 96.987, 25.793, -1.714]
  MoveL 3878 to (-45.77, 29.43, -120.13) mm, rotated rx -167.81 ry 3.47 rz -52.11 deg; joints [2.109, -28.967, 98.634, 148.565, 97.088, 25.71, -1.714]
  MoveL 3879 to (-46.85, 27.29, -119.94) mm, rotated rx -167.81 ry 3.47 rz -52.11 deg; joints [2.159, -29, 98.802, 148.601, 97.195, 25.624, -1.714]
  MoveL 3880 to (-47.9, 25.21, -119.74) mm, rotated rx -167.81 ry 3.47 rz -52.11 deg; joints [2.207, -29.03, 98.965, 148.636, 97.299, 25.541, -1.714]
  MoveL 3881 to (-48.86, 23.3, -119.62) mm, rotated rx -167.81 ry 3.47 rz -52.11 deg; joints [2.251, -29.062, 99.116, 148.667, 97.394, 25.465, -1.714]
  MoveL 3882 to (-50.75, 19.52, -119.35) mm, rotated rx -167.81 ry 3.47 rz -52.11 deg; joints [2.338, -29.12, 99.414, 148.729, 97.583, 25.314, -1.714]
  MoveL 3883 to (-51.72, 17.58, -119.29) mm, rotated rx -167.81 ry 3.47 rz -52.11 deg; joints [2.382, -29.155, 99.571, 148.76, 97.679, 25.238, -1.714]
  MoveL 3884 to (-52.66, 15.66, -119.06) mm, rotated rx -167.81 ry 3.47 rz -52.11 deg; joints [2.426, -29.179, 99.716, 148.792, 97.776, 25.161, -1.714]
  MoveL 3885 to (-53.59, 13.77, -118.9) mm, rotated rx -167.81 ry 3.47 rz -52.11 deg; joints [2.47, -29.205, 99.862, 148.823, 97.871, 25.086, -1.714]
  MoveL 3886 to (-54.51, 11.87, -118.72) mm, rotated rx -167.81 ry 3.47 rz -52.11 deg; joints [2.513, -29.23, 100.007, 148.853, 97.966, 25.011, -1.714]
  MoveL 3887 to (-55.48, 9.92, -118.63) mm, rotated rx -167.81 ry 3.47 rz -52.11 deg; joints [2.558, -29.262, 100.162, 148.885, 98.063, 24.934, -1.714]
  MoveL 3888 to (-56.47, 7.87, -118.5) mm, rotated rx -167.81 ry 3.47 rz -52.11 deg; joints [2.604, -29.293, 100.321, 148.917, 98.166, 24.854, -1.714]
  MoveL 3889 to (-57.34, 6.18, -118.44) mm, rotated rx -167.81 ry 3.47 rz -52.11 deg; joints [2.644, -29.322, 100.456, 148.945, 98.25, 24.788, -1.714]
  MoveL 3890 to (-56.74, 5.88, -117.56) mm, rotated rx -167.81 ry 3.47 rz -52.11 deg; joints [2.633, -29.257, 100.425, 148.933, 98.28, 24.773, -1.714]
  MoveL 3891 to (-56.42, 6.04, -117.14) mm, rotated rx -167.81 ry 3.47 rz -52.11 deg; joints [2.626, -29.223, 100.387, 148.926, 98.278, 24.778, -1.714]
  MoveL 3892 to (-56.35, 6.03, -116.86) mm, rotated rx -167.81 ry 3.47 rz -52.11 deg; joints [2.626, -29.204, 100.371, 148.927, 98.281, 24.776, -1.714]
  MoveL 3893 to (-56.61, 5.82, -116.75) mm, rotated rx -167.81 ry 3.47 rz -52.11 deg; joints [2.638, -29.203, 100.382, 148.936, 98.289, 24.766, -1.714]
  MoveL 3894 to (-56.98, 5.57, -116.69) mm, rotated rx -167.81 ry 3.47 rz -52.11 deg; joints [2.653, -29.209, 100.401, 148.949, 98.298, 24.755, -1.714]
  MoveL 3895 to (-57.46, 5.27, -116.65) mm, rotated rx -167.81 ry 3.47 rz -52.11 deg; joints [2.672, -29.218, 100.426, 148.965, 98.308, 24.742, -1.714]
  MoveL 3896 to (-58.06, 4.91, -116.61) mm, rotated rx -167.81 ry 3.47 rz -52.11 deg; joints [2.696, -29.23, 100.457, 148.986, 98.32, 24.725, -1.714]
  MoveL 3897 to (-58.6, 4.59, -116.59) mm, rotated rx -167.81 ry 3.47 rz -52.11 deg; joints [2.717, -29.242, 100.484, 149.004, 98.331, 24.711, -1.714]
  MoveL 3898 to (-59.06, 4.34, -116.59) mm, rotated rx -167.81 ry 3.47 rz -52.11 deg; joints [2.735, -29.253, 100.508, 149.019, 98.338, 24.699, -1.714]
  MoveL 3899 to (-59.48, 4.09, -116.57) mm, rotated rx -167.81 ry 3.47 rz -52.11 deg; joints [2.752, -29.262, 100.529, 149.033, 98.346, 24.688, -1.714]
  MoveL 3900 to (-60.36, 3.53, -116.49) mm, rotated rx -167.81 ry 3.47 rz -52.11 deg; joints [2.787, -29.278, 100.575, 149.063, 98.365, 24.663, -1.714]
  MoveL 3901 to (-60.83, 3.23, -116.45) mm, rotated rx -167.81 ry 3.47 rz -52.11 deg; joints [2.806, -29.287, 100.599, 149.079, 98.376, 24.65, -1.714]
  MoveL 3902 to (-61.25, 2.94, -116.38) mm, rotated rx -167.81 ry 3.47 rz -52.11 deg; joints [2.824, -29.293, 100.621, 149.094, 98.386, 24.637, -1.714]
  MoveL 3903 to (-61.63, 2.67, -116.3) mm, rotated rx -167.81 ry 3.47 rz -52.11 deg; joints [2.84, -29.297, 100.64, 149.107, 98.396, 24.625, -1.714]
  MoveL 3904 to (-62.01, 2.41, -116.25) mm, rotated rx -167.81 ry 3.47 rz -52.11 deg; joints [2.855, -29.303, 100.66, 149.12, 98.406, 24.613, -1.714]
  MoveL 3905 to (-62.42, 2.15, -116.21) mm, rotated rx -167.81 ry 3.47 rz -52.11 deg; joints [2.872, -29.311, 100.681, 149.134, 98.414, 24.602, -1.714]
  MoveL 3906 to (-62.87, 1.88, -116.19) mm, rotated rx -167.81 ry 3.47 rz -52.11 deg; joints [2.89, -29.321, 100.704, 149.15, 98.423, 24.59, -1.714]
  MoveL 3907 to (-66.07, 0.09, -116.19) mm, rotated rx -167.81 ry 3.47 rz -52.11 deg; joints [3.015, -29.396, 100.866, 149.256, 98.477, 24.511, -1.714]
  MoveL 3908 to (-67.54, -0.61, -116.22) mm, rotated rx -167.81 ry 3.47 rz -52.11 deg; joints [3.072, -29.431, 100.932, 149.306, 98.494, 24.479, -1.714]
  MoveL 3909 to (-68.09, -0.77, -116.24) mm, rotated rx -167.81 ry 3.47 rz -52.11 deg; joints [3.092, -29.444, 100.949, 149.324, 98.495, 24.471, -1.714]
  MoveL 3910 to (-68.53, -0.82, -116.28) mm, rotated rx -167.81 ry 3.47 rz -52.11 deg; joints [3.108, -29.455, 100.958, 149.338, 98.491, 24.467, -1.714]
